    robot6axis_ctrled1/robot6axis/servo_2/servo_control/OperationMode AT 677 : INT := 0;
    robot6axis_ctrled1/robot6axis/servo_2/servo_control/StatusReady AT 253 : BOOL := true;
    robot6axis_ctrled1/robot6axis/servo_2/servo_control/StatusMove AT 254 : BOOL := false;
    robot6axis_ctrled1/robot6axis/servo_2/servo_control/StatusStand AT 255 : BOOL := false;
    robot6axis_ctrled1/robot6axis/servo_2/servo_control/ActualPositionMa AT 6703 : REAL := 0.0;
    robot6axis_ctrled1/robot6axis/servo_2/servo_control/ActualVelocity AT 6704 : REAL := 0.0;
    robot6axis_ctrled1/robot6axis/servo_2/servo_control/MaximumVelocity AT 6705 : REAL := 0.0;
    robot6axis_ctrled1/robot6axis/servo_2/servo_control/VelEnabled AT 256 : BOOL := false;
    robot6axis_ctrled1/robot6axis/servo_2/servo_control/VelCmd AT 257 : BOOL := false;
    robot6axis_ctrled1/robot6axis/servo_2/servo_control/PosEnabled AT 258 : BOOL := false;
    robot6axis_ctrled1/robot6axis/servo_2/servo_control/PosCmd AT 259 : BOOL := false;
    robot6axis_ctrled1/robot6axis/servo_2/servo_control/Position AT 6707 : REAL := 0.0;
    robot6axis_ctrled1/robot6axis/servo_2/servo_control/Speed AT 6706 : REAL := 0.0;
    robot6axis_ctrled1/robot6axis/servo_2/servo_control/ManualMode AT 678 : INT := 0;
    robot6axis_ctrled1/robot6axis/servo_2/servo_control/initDone AT 263 : BOOL := false;
    robot6axis_ctrled1/robot6axis/servo_2/servo_control/ActualPositionMa1 AT 6717 : REAL := 0.0;
    robot6axis_ctrled1/robot6axis/servo_2/servo_control/offsetAxToMa1 AT 6718 : REAL := 0.0;
    robot6axis_ctrled1/robot6axis/servo_2/servo_control/HOME_POSITION AT 6719 : REAL := 100.0;
    robot6axis_ctrled1/robot6axis/servo_2/servo_control/MANUAL_POSITION1 AT 6720 : REAL := 0.0;
    robot6axis_ctrled1/robot6axis/servo_2/servo_control/MANUAL_POSITION2 AT 6721 : REAL := 150.0;
    robot6axis_ctrled1/robot6axis/servo_2/servo_control/MANUAL_SPEED1 AT 6722 : REAL := -100.0;
    robot6axis_ctrled1/robot6axis/servo_2/servo_control/MANUAL_SPEED2 AT 6723 : REAL := 100.0;
    robot6axis_ctrled1/robot6axis/servo_2/servo_control/MANUAL_SPEED AT 6724 : REAL := 100.0;
    robot6axis_ctrled1/robot6axis/servo_2/servo_velocity/MoveVelEnable AT 256 : BOOL := false;
    robot6axis_ctrled1/robot6axis/servo_2/servo_velocity/MoveVelStart AT 257 : BOOL := false;
    robot6axis_ctrled1/robot6axis/servo_2/servo_velocity/MoveSpeed AT 6706 : REAL := 0.0;
    robot6axis_ctrled1/robot6axis/servo_2/servo_velocity/MoveAcceleration AT 86 : REAL := 100.0;
    robot6axis_ctrled1/robot6axis/servo_2/servo_velocity/MoveDeceleration AT 85 : REAL := 100.0;
    robot6axis_ctrled1/robot6axis/servo_2/servo_velocity/MAX_SPEED AT 6499 : REAL(0.0..3.4e+038) := 30.0;
    robot6axis_ctrled1/robot6axis/servo_2/servo_velocity/MAX_ACCEL AT 6498 : REAL(0.0..3.4e+038) := 1500.0;
    robot6axis_ctrled1/robot6axis/servo_2/servo_velocity/MAX_DECEL AT 6497 : REAL(0.0..3.4e+038) := 1500.0;
    robot6axis_ctrled1/robot6axis/servo_2/servo_velocity/MODULO_LENGTH AT 6496 : REAL := 0.0;
    robot6axis_ctrled1/robot6axis/servo_2/servo_velocity/status AT 661 : INT := 0;
    robot6axis_ctrled1/robot6axis/servo_2/servo_velocity/errorFlag AT 660 : INT := 0;
    robot6axis_ctrled1/robot6axis/servo_2/servo_velocity/MoveVelDone AT 225 : BOOL := false;
    robot6axis_ctrled1/robot6axis/servo_2/servo_velocity/ActualPositionAx AT 6502 : REAL := 0.0;
    robot6axis_ctrled1/robot6axis/servo_2/servo_velocity/ActualVelocity AT 6501 : REAL := 0.0;
    robot6axis_ctrled1/robot6axis/servo_2/servo_velocity/firstStep AT 264 : BOOL := true;
    robot6axis_ctrled1/robot6axis/servo_2/servo_velocity/stepDone AT 265 : BOOL := false;
    robot6axis_ctrled1/robot6axis/servo_2/servo_velocity/currentTime AT 6725 : REAL := 0.0;
    robot6axis_ctrled1/robot6axis/servo_2/servo_velocity/MoveSpeed1 AT 6726 : REAL := 0.0;
    robot6axis_ctrled1/robot6axis/servo_2/servo_velocity/acceleration AT 6727 : REAL := 0.0;
    robot6axis_ctrled1/robot6axis/servo_2/servo_velocity/deceleration AT 6728 : REAL := 0.0;
    robot6axis_ctrled1/robot6axis/servo_2/servo_velocity/orderSpeed AT 6729 : REAL := 0.0;
    robot6axis_ctrled1/robot6axis/servo_2/servo_velocity/endChangeSpeed AT 6730 : REAL := 0.0;
    robot6axis_ctrled1/robot6axis/servo_2/servo_velocity/accelDecelChangeSpeed AT 6731 : REAL := 0.0;
    robot6axis_ctrled1/robot6axis/servo_2/servo_velocity/ActualVelocity1 AT 6732 : REAL := 0.0;
    robot6axis_ctrled1/robot6axis/servo_2/servo_velocity/speedChanged AT 266 : BOOL := false;
    robot6axis_ctrled1/robot6axis/servo_2/servo_position/MoveAbsEnable AT 258 : BOOL := false;
    robot6axis_ctrled1/robot6axis/servo_2/servo_position/MoveAbsStart AT 259 : BOOL := false;
    robot6axis_ctrled1/robot6axis/servo_2/servo_position/MovePosition AT 6707 : REAL := 0.0;
    robot6axis_ctrled1/robot6axis/servo_2/servo_position/MoveSpeed AT 6706 : REAL := 0.0;
    robot6axis_ctrled1/robot6axis/servo_2/servo_position/MoveAcceleration AT 86 : REAL := 100.0;
    robot6axis_ctrled1/robot6axis/servo_2/servo_position/MoveDeceleration AT 85 : REAL := 100.0;
    robot6axis_ctrled1/robot6axis/servo_2/servo_position/MAX_SPEED AT 6499 : REAL(0.0..3.4e+038) := 30.0;
    robot6axis_ctrled1/robot6axis/servo_2/servo_position/MAX_ACCEL AT 6498 : REAL(0.0..3.4e+038) := 1500.0;
    robot6axis_ctrled1/robot6axis/servo_2/servo_position/MAX_DECEL AT 6497 : REAL(0.0..3.4e+038) := 1500.0;
    robot6axis_ctrled1/robot6axis/servo_2/servo_position/MODULO_LENGTH AT 6496 : REAL := 0.0;
    robot6axis_ctrled1/robot6axis/servo_2/servo_position/status AT 661 : INT := 0;
    robot6axis_ctrled1/robot6axis/servo_2/servo_position/errorFlag AT 660 : INT := 0;
    robot6axis_ctrled1/robot6axis/servo_2/servo_position/MoveAbsDone AT 224 : BOOL := false;
    robot6axis_ctrled1/robot6axis/servo_2/servo_position/ActualPositionAx AT 6502 : REAL := 0.0;
    robot6axis_ctrled1/robot6axis/servo_2/servo_position/ActualVelocity AT 6501 : REAL := 0.0;
    robot6axis_ctrled1/robot6axis/servo_2/servo_position/firstStep AT 267 : BOOL := true;
    robot6axis_ctrled1/robot6axis/servo_2/servo_position/stepDone AT 268 : BOOL := false;
    robot6axis_ctrled1/robot6axis/servo_2/servo_position/timeToStop AT 6733 : REAL := 0.0;
    robot6axis_ctrled1/robot6axis/servo_2/servo_position/distanceToStop AT 6734 : REAL := 0.0;
    robot6axis_ctrled1/robot6axis/servo_2/servo_position/distance AT 6735 : REAL := 0.0;
    robot6axis_ctrled1/robot6axis/servo_2/servo_position/currentTime AT 6736 : REAL := 0.0;
    robot6axis_ctrled1/robot6axis/servo_2/servo_position/currentSpeed1 AT 6737 : REAL := 0.0;
    robot6axis_ctrled1/robot6axis/servo_2/servo_position/targetPosition AT 6738 : REAL := 0.0;
    robot6axis_ctrled1/robot6axis/servo_2/servo_position/ActualPositionAx1 AT 6739 : REAL := 0.0;
    robot6axis_ctrled1/robot6axis/servo_2/servo_position/acceleration AT 6740 : REAL := 0.0;
    robot6axis_ctrled1/robot6axis/servo_2/servo_position/deceleration AT 6741 : REAL := 0.0;
    robot6axis_ctrled1/robot6axis/servo_2/servo_position/orderSpeed AT 6742 : REAL := 0.0;
    robot6axis_ctrled1/robot6axis/servo_2/servo_position/moveDirection AT 6743 : REAL := 0.0;
    robot6axis_ctrled1/robot6axis/servo_2/servo_position/moveDirection1 AT 6744 : REAL := 0.0;
    robot6axis_ctrled1/robot6axis/servo_2/servo_position/endChangeSpeed AT 6745 : REAL := 0.0;
    robot6axis_ctrled1/robot6axis/servo_2/servo_position/ActualVelocity1 AT 6746 : REAL := 0.0;
    robot6axis_ctrled1/robot6axis/arm2/armOrigin AT 6540 : ARRAY[1..3] OF REAL := [3(0.0)];
    robot6axis_ctrled1/robot6axis/arm2/overallArmQuatInput AT 6545 : ARRAY[1..4] OF REAL := [4(0.0)];
    robot6axis_ctrled1/robot6axis/arm2/structRotVector AT 149 : ARRAY[1..3] OF REAL := [2(0.0), 1.0];
    robot6axis_ctrled1/robot6axis/arm2/structRotDeg AT 148 : REAL := -90.0;
    robot6axis_ctrled1/robot6axis/arm2/driveRotVector AT 138 : ARRAY[1..3] OF REAL := [0.0, 1.0, 0.0];
    robot6axis_ctrled1/robot6axis/arm2/driveRotDeg AT 6551 : REAL := 0.0;
    robot6axis_ctrled1/robot6axis/arm2/ownRotDeg AT 6492 : REAL := 0.0;
    robot6axis_ctrled1/robot6axis/arm2/driveResizeLength AT 6491 : REAL := 0.0;
    robot6axis_ctrled1/robot6axis/arm2/functionActive AT 218 : BOOL := false;
    robot6axis_ctrled1/robot6axis/arm2/armExtrem AT 6552 : ARRAY[1..3] OF REAL := [3(0.0)];
    robot6axis_ctrled1/robot6axis/arm2/overallArmRotOutput AT 6557 : ARRAY[1..4] OF REAL := [4(0.0)];
    robot6axis_ctrled1/robot6axis/arm2/productId AT 659 : DINT := -1;
    robot6axis_ctrled1/robot6axis/arm2/status_act_prod AT 679 : DINT := 0;
    robot6axis_ctrled1/robot6axis/arm2/m11 AT 6747 : REAL := 127.321;
    robot6axis_ctrled1/robot6axis/arm2/m12 AT 6748 : REAL := 0.0;
    robot6axis_ctrled1/robot6axis/arm2/m13 AT 6749 : REAL := 0.0;
    robot6axis_ctrled1/robot6axis/arm2/m14 AT 6750 : REAL := 453.404;
    robot6axis_ctrled1/robot6axis/arm2/m21 AT 6751 : REAL := 0.0;
    robot6axis_ctrled1/robot6axis/arm2/m22 AT 6752 : REAL := 1.0;
    robot6axis_ctrled1/robot6axis/arm2/m23 AT 6753 : REAL := 0.0;
    robot6axis_ctrled1/robot6axis/arm2/m24 AT 6754 : REAL := 1.0;
    robot6axis_ctrled1/robot6axis/arm2/m31 AT 6755 : REAL := 0.0;
    robot6axis_ctrled1/robot6axis/arm2/m32 AT 6756 : REAL := 0.0;
    robot6axis_ctrled1/robot6axis/arm2/m33 AT 6757 : REAL := 35.3669;
    robot6axis_ctrled1/robot6axis/arm2/m34 AT 6758 : REAL := 213.705;
    robot6axis_ctrled1/robot6axis/arm2/m41 AT 6759 : REAL := 0.0;
    robot6axis_ctrled1/robot6axis/arm2/m42 AT 6760 : REAL := 0.0;
    robot6axis_ctrled1/robot6axis/arm2/m43 AT 6761 : REAL := 0.0;
    robot6axis_ctrled1/robot6axis/arm2/m44 AT 6762 : REAL := 1.0;
    robot6axis_ctrled1/robot6axis/arm2/armLengthCalc AT 6763 : REAL := 0.0;
    robot6axis_ctrled1/robot6axis/arm2/functionActiveLocale AT 269 : BOOL := false;
    robot6axis_ctrled1/robot6axis/arm2/product_id AT 680 : DINT := -1;
    robot6axis_ctrled1/robot6axis/arm2/arm_id AT 681 : DINT := -1;
    robot6axis_ctrled1/robot6axis/arm2/timeToGripParam AT 6764 : REAL := 0.15;
    robot6axis_ctrled1/robot6axis/arm2/armLength AT 6765 : REAL := 290.0;
    robot6axis_ctrled1/robot6axis/arm2/armWidth AT 6766 : REAL := 60.0;
    robot6axis_ctrled1/robot6axis/arm2/armHeight AT 6767 : REAL := 60.0;
    robot6axis_ctrled1/robot6axis/arm2/armType AT 682 : INT := 0;
    robot6axis_ctrled1/robot6axis/servo_3/status AT 658 : INT := 0;
    robot6axis_ctrled1/robot6axis/servo_3/errorFlag AT 657 : INT := 0;
    robot6axis_ctrled1/robot6axis/servo_3/ActualPositionAx1 AT 6490 : REAL := 0.0;
    robot6axis_ctrled1/robot6axis/servo_3/MoveVelDone1 AT 217 : BOOL := false;
    robot6axis_ctrled1/robot6axis/servo_3/ActualVelocity1 AT 6489 : REAL := 0.0;
    robot6axis_ctrled1/robot6axis/servo_3/MoveAbsDone1 AT 216 : BOOL := false;
    robot6axis_ctrled1/robot6axis/servo_3/HomeCmd AT 84 : BOOL := false;
    robot6axis_ctrled1/robot6axis/servo_3/MoveVelCmd AT 83 : BOOL := false;
    robot6axis_ctrled1/robot6axis/servo_3/MoveAbsCmd AT 82 : BOOL := false;
    robot6axis_ctrled1/robot6axis/servo_3/MoveVel1ManualCmd AT 81 : BOOL := false;
    robot6axis_ctrled1/robot6axis/servo_3/MoveVel2ManualCmd AT 80 : BOOL := false;
    robot6axis_ctrled1/robot6axis/servo_3/MoveAbs1ManualCmd AT 79 : BOOL := false;
    robot6axis_ctrled1/robot6axis/servo_3/MoveAbs2ManualCmd AT 78 : BOOL := false;
    robot6axis_ctrled1/robot6axis/servo_3/StopCmd AT 22 : BOOL := false;
    robot6axis_ctrled1/robot6axis/servo_3/MovePosition AT 83 : REAL := 0.0;
    robot6axis_ctrled1/robot6axis/servo_3/MoveSpeed AT 82 : REAL := 100.0;
    robot6axis_ctrled1/robot6axis/servo_3/MoveAcceleration AT 81 : REAL := 100.0;
    robot6axis_ctrled1/robot6axis/servo_3/MoveDeceleration AT 80 : REAL := 100.0;
    robot6axis_ctrled1/robot6axis/servo_3/offsetAxToMa AT 79 : REAL := 0.0;
    robot6axis_ctrled1/robot6axis/servo_3/PLC_StatusReady AT 50 : BOOL := true;
    robot6axis_ctrled1/robot6axis/servo_3/PLC_StatusMoved AT 49 : BOOL := false;
    robot6axis_ctrled1/robot6axis/servo_3/PLC_StatusStand AT 48 : BOOL := false;
    robot6axis_ctrled1/robot6axis/servo_3/PLC_ActualPositionAx AT 169 : REAL := 0.0;
    robot6axis_ctrled1/robot6axis/servo_3/PLC_ActualPositionMa AT 59 : REAL := 0.0;
    robot6axis_ctrled1/robot6axis/servo_3/PLC_ActualVelocity AT 58 : REAL := 0.0;
    robot6axis_ctrled1/robot6axis/servo_3/physicalPosInit AT 6488 : REAL := 0.0;
    robot6axis_ctrled1/robot6axis/servo_3/MAX_SPEED AT 6487 : REAL(0.0..3.4e+038) := 30.0;
    robot6axis_ctrled1/robot6axis/servo_3/MAX_ACCEL AT 6486 : REAL(0.0..3.4e+038) := 1500.0;
    robot6axis_ctrled1/robot6axis/servo_3/MAX_DECEL AT 6485 : REAL(0.0..3.4e+038) := 1500.0;
    robot6axis_ctrled1/robot6axis/servo_3/MODULO_LENGTH AT 6484 : REAL := 0.0;
    robot6axis_ctrled1/robot6axis/servo_3/StatusReady AT 215 : BOOL := true;
    robot6axis_ctrled1/robot6axis/servo_3/StatusMoved AT 214 : BOOL := false;
    robot6axis_ctrled1/robot6axis/servo_3/StatusStand AT 213 : BOOL := false;
    robot6axis_ctrled1/robot6axis/servo_3/ActualPositionAx AT 6563 : REAL := 0.0;
    robot6axis_ctrled1/robot6axis/servo_3/ActualPositionMa AT 6483 : REAL := 0.0;
    robot6axis_ctrled1/robot6axis/servo_3/ActualVelocity AT 49 : REAL := 0.0;
    robot6axis_ctrled1/robot6axis/servo_3/MaximumVelocity AT 6482 : REAL := 0.0;
    robot6axis_ctrled1/robot6axis/servo_3/StatusPosIncrease AT 212 : BOOL := false;
    robot6axis_ctrled1/robot6axis/servo_3/StatusPosDecrease AT 211 : BOOL := false;
    robot6axis_ctrled1/robot6axis/servo_3/displayJauge AT 6481 : REAL := 0.0;
    robot6axis_ctrled1/robot6axis/servo_3/servo_mode/PLC_StatusReady AT 50 : BOOL := true;
    robot6axis_ctrled1/robot6axis/servo_3/servo_mode/PLC_StatusMoved AT 49 : BOOL := false;
    robot6axis_ctrled1/robot6axis/servo_3/servo_mode/PLC_StatusStand AT 48 : BOOL := false;
    robot6axis_ctrled1/robot6axis/servo_3/servo_mode/PLC_ActualPositionAx AT 169 : REAL := 0.0;
    robot6axis_ctrled1/robot6axis/servo_3/servo_mode/PLC_ActualPositionMa AT 59 : REAL := 0.0;
    robot6axis_ctrled1/robot6axis/servo_3/servo_mode/PLC_ActualVelocity AT 58 : REAL := 0.0;
    robot6axis_ctrled1/robot6axis/servo_3/servo_mode/StatusReady AT 270 : BOOL := true;
    robot6axis_ctrled1/robot6axis/servo_3/servo_mode/StatusMoved AT 271 : BOOL := false;
    robot6axis_ctrled1/robot6axis/servo_3/servo_mode/StatusStand AT 272 : BOOL := false;
    robot6axis_ctrled1/robot6axis/servo_3/servo_mode/ActualPositionMa AT 6768 : REAL := 0.0;
    robot6axis_ctrled1/robot6axis/servo_3/servo_mode/ActualVelocity AT 6769 : REAL := 0.0;
    robot6axis_ctrled1/robot6axis/servo_3/servo_mode/MaximumVelocity AT 6770 : REAL := 0.0;
    robot6axis_ctrled1/robot6axis/servo_3/servo_mode/physicalPosInit AT 6488 : REAL := 0.0;
    robot6axis_ctrled1/robot6axis/servo_3/servo_mode/ActualPositionAx AT 6490 : REAL := 0.0;
    robot6axis_ctrled1/robot6axis/servo_3/servo_mode/StatusReady_o AT 215 : BOOL := true;
    robot6axis_ctrled1/robot6axis/servo_3/servo_mode/StatusMoved_o AT 214 : BOOL := false;
    robot6axis_ctrled1/robot6axis/servo_3/servo_mode/StatusStand_o AT 213 : BOOL := false;
    robot6axis_ctrled1/robot6axis/servo_3/servo_mode/ActualPositionAx_o AT 6563 : REAL := 0.0;
    robot6axis_ctrled1/robot6axis/servo_3/servo_mode/ActualPositionMa_o AT 6483 : REAL := 0.0;
    robot6axis_ctrled1/robot6axis/servo_3/servo_mode/ActualVelocity_o AT 49 : REAL := 0.0;
    robot6axis_ctrled1/robot6axis/servo_3/servo_mode/MaximumVelocity_o AT 6482 : REAL := 0.0;
    robot6axis_ctrled1/robot6axis/servo_3/servo_mode/StatusPosIncrease_o AT 212 : BOOL := false;
    robot6axis_ctrled1/robot6axis/servo_3/servo_mode/StatusPosDecrease_o AT 211 : BOOL := false;
    robot6axis_ctrled1/robot6axis/servo_3/servo_mode/displayJauge_o AT 6481 : REAL := 0.0;
    robot6axis_ctrled1/robot6axis/servo_3/servo_mode/PLCMode AT 277 : BOOL := false;
    robot6axis_ctrled1/robot6axis/servo_3/servo_mode/PLCMode1 AT 278 : BOOL := false;
    robot6axis_ctrled1/robot6axis/servo_3/servo_mode/initDone AT 279 : BOOL := false;
    robot6axis_ctrled1/robot6axis/servo_3/servo_mode/displayPosMin AT 6773 : REAL := 0.0;
    robot6axis_ctrled1/robot6axis/servo_3/servo_mode/displayPosMax AT 6774 : REAL := 0.0;
    robot6axis_ctrled1/robot6axis/servo_3/servo_mode/PLC_ActualPositionAx1 AT 6775 : REAL := 0.0;
    robot6axis_ctrled1/robot6axis/servo_3/servo_mode/PLC_ActualVelocity1 AT 6776 : REAL := 0.0;
    robot6axis_ctrled1/robot6axis/servo_3/servo_mode/ActualPositionAx1 AT 6777 : REAL := 0.0;
    robot6axis_ctrled1/robot6axis/servo_3/servo_mode/ActualVelocity1 AT 6778 : REAL := 0.0;
    robot6axis_ctrled1/robot6axis/servo_3/servo_mode/offsetAxToMa AT 6779 : REAL := 0.0;
    robot6axis_ctrled1/robot6axis/servo_3/servo_mode/offsetAxToMa1 AT 6780 : REAL := 0.0;
    robot6axis_ctrled1/robot6axis/servo_3/servo_mode/ActualPositionMa_o1 AT 6781 : REAL := 0.0;
    robot6axis_ctrled1/robot6axis/servo_3/servo_control/HomeCmd AT 84 : BOOL := false;
    robot6axis_ctrled1/robot6axis/servo_3/servo_control/MoveVelCmd AT 83 : BOOL := false;
    robot6axis_ctrled1/robot6axis/servo_3/servo_control/MoveAbsCmd AT 82 : BOOL := false;
    robot6axis_ctrled1/robot6axis/servo_3/servo_control/MoveVel1ManualCmd AT 81 : BOOL := false;
    robot6axis_ctrled1/robot6axis/servo_3/servo_control/MoveVel2ManualCmd AT 80 : BOOL := false;
    robot6axis_ctrled1/robot6axis/servo_3/servo_control/MoveAbs1ManualCmd AT 79 : BOOL := false;
    robot6axis_ctrled1/robot6axis/servo_3/servo_control/MoveAbs2ManualCmd AT 78 : BOOL := false;
    robot6axis_ctrled1/robot6axis/servo_3/servo_control/StopCmd AT 22 : BOOL := false;
    robot6axis_ctrled1/robot6axis/servo_3/servo_control/MovePosition AT 83 : REAL := 0.0;
    robot6axis_ctrled1/robot6axis/servo_3/servo_control/MoveSpeed AT 82 : REAL := 100.0;
    robot6axis_ctrled1/robot6axis/servo_3/servo_control/MoveAcceleration AT 81 : REAL := 100.0;
    robot6axis_ctrled1/robot6axis/servo_3/servo_control/MoveDeceleration AT 80 : REAL := 100.0;
    robot6axis_ctrled1/robot6axis/servo_3/servo_control/offsetAxToMa AT 79 : REAL := 0.0;
    robot6axis_ctrled1/robot6axis/servo_3/servo_control/physicalPosInit AT 6488 : REAL := 0.0;
    robot6axis_ctrled1/robot6axis/servo_3/servo_control/MAX_SPEED AT 6487 : REAL(0.0..3.4e+038) := 30.0;
    robot6axis_ctrled1/robot6axis/servo_3/servo_control/status AT 658 : INT := 0;
    robot6axis_ctrled1/robot6axis/servo_3/servo_control/errorFlag AT 657 : INT := 0;
    robot6axis_ctrled1/robot6axis/servo_3/servo_control/IOActualPositionAx AT 6490 : REAL := 0.0;
    robot6axis_ctrled1/robot6axis/servo_3/servo_control/IOVelDone AT 217 : BOOL := false;
    robot6axis_ctrled1/robot6axis/servo_3/servo_control/IOAbsDone AT 216 : BOOL := false;
    robot6axis_ctrled1/robot6axis/servo_3/servo_control/IOActualVelocity AT 6489 : REAL := 0.0;
    robot6axis_ctrled1/robot6axis/servo_3/servo_control/OperationMode AT 683 : INT := 0;
    robot6axis_ctrled1/robot6axis/servo_3/servo_control/StatusReady AT 270 : BOOL := true;
    robot6axis_ctrled1/robot6axis/servo_3/servo_control/StatusMove AT 271 : BOOL := false;
    robot6axis_ctrled1/robot6axis/servo_3/servo_control/StatusStand AT 272 : BOOL := false;
    robot6axis_ctrled1/robot6axis/servo_3/servo_control/ActualPositionMa AT 6768 : REAL := 0.0;
    robot6axis_ctrled1/robot6axis/servo_3/servo_control/ActualVelocity AT 6769 : REAL := 0.0;
    robot6axis_ctrled1/robot6axis/servo_3/servo_control/MaximumVelocity AT 6770 : REAL := 0.0;
    robot6axis_ctrled1/robot6axis/servo_3/servo_control/VelEnabled AT 273 : BOOL := false;
    robot6axis_ctrled1/robot6axis/servo_3/servo_control/VelCmd AT 274 : BOOL := false;
    robot6axis_ctrled1/robot6axis/servo_3/servo_control/PosEnabled AT 275 : BOOL := false;
    robot6axis_ctrled1/robot6axis/servo_3/servo_control/PosCmd AT 276 : BOOL := false;
    robot6axis_ctrled1/robot6axis/servo_3/servo_control/Position AT 6772 : REAL := 0.0;
    robot6axis_ctrled1/robot6axis/servo_3/servo_control/Speed AT 6771 : REAL := 0.0;
    robot6axis_ctrled1/robot6axis/servo_3/servo_control/ManualMode AT 684 : INT := 0;
    robot6axis_ctrled1/robot6axis/servo_3/servo_control/initDone AT 280 : BOOL := false;
    robot6axis_ctrled1/robot6axis/servo_3/servo_control/ActualPositionMa1 AT 6782 : REAL := 0.0;
    robot6axis_ctrled1/robot6axis/servo_3/servo_control/offsetAxToMa1 AT 6783 : REAL := 0.0;
    robot6axis_ctrled1/robot6axis/servo_3/servo_control/HOME_POSITION AT 6784 : REAL := 100.0;
    robot6axis_ctrled1/robot6axis/servo_3/servo_control/MANUAL_POSITION1 AT 6785 : REAL := 0.0;
    robot6axis_ctrled1/robot6axis/servo_3/servo_control/MANUAL_POSITION2 AT 6786 : REAL := 150.0;
    robot6axis_ctrled1/robot6axis/servo_3/servo_control/MANUAL_SPEED1 AT 6787 : REAL := -100.0;
    robot6axis_ctrled1/robot6axis/servo_3/servo_control/MANUAL_SPEED2 AT 6788 : REAL := 100.0;
    robot6axis_ctrled1/robot6axis/servo_3/servo_control/MANUAL_SPEED AT 6789 : REAL := 100.0;
    robot6axis_ctrled1/robot6axis/servo_3/servo_velocity/MoveVelEnable AT 273 : BOOL := false;
    robot6axis_ctrled1/robot6axis/servo_3/servo_velocity/MoveVelStart AT 274 : BOOL := false;
    robot6axis_ctrled1/robot6axis/servo_3/servo_velocity/MoveSpeed AT 6771 : REAL := 0.0;
    robot6axis_ctrled1/robot6axis/servo_3/servo_velocity/MoveAcceleration AT 81 : REAL := 100.0;
    robot6axis_ctrled1/robot6axis/servo_3/servo_velocity/MoveDeceleration AT 80 : REAL := 100.0;
    robot6axis_ctrled1/robot6axis/servo_3/servo_velocity/MAX_SPEED AT 6487 : REAL(0.0..3.4e+038) := 30.0;
    robot6axis_ctrled1/robot6axis/servo_3/servo_velocity/MAX_ACCEL AT 6486 : REAL(0.0..3.4e+038) := 1500.0;
    robot6axis_ctrled1/robot6axis/servo_3/servo_velocity/MAX_DECEL AT 6485 : REAL(0.0..3.4e+038) := 1500.0;
    robot6axis_ctrled1/robot6axis/servo_3/servo_velocity/MODULO_LENGTH AT 6484 : REAL := 0.0;
    robot6axis_ctrled1/robot6axis/servo_3/servo_velocity/status AT 658 : INT := 0;
    robot6axis_ctrled1/robot6axis/servo_3/servo_velocity/errorFlag AT 657 : INT := 0;
    robot6axis_ctrled1/robot6axis/servo_3/servo_velocity/MoveVelDone AT 217 : BOOL := false;
    robot6axis_ctrled1/robot6axis/servo_3/servo_velocity/ActualPositionAx AT 6490 : REAL := 0.0;
    robot6axis_ctrled1/robot6axis/servo_3/servo_velocity/ActualVelocity AT 6489 : REAL := 0.0;
    robot6axis_ctrled1/robot6axis/servo_3/servo_velocity/firstStep AT 281 : BOOL := true;
    robot6axis_ctrled1/robot6axis/servo_3/servo_velocity/stepDone AT 282 : BOOL := false;
    robot6axis_ctrled1/robot6axis/servo_3/servo_velocity/currentTime AT 6790 : REAL := 0.0;
    robot6axis_ctrled1/robot6axis/servo_3/servo_velocity/MoveSpeed1 AT 6791 : REAL := 0.0;
    robot6axis_ctrled1/robot6axis/servo_3/servo_velocity/acceleration AT 6792 : REAL := 0.0;
    robot6axis_ctrled1/robot6axis/servo_3/servo_velocity/deceleration AT 6793 : REAL := 0.0;
    robot6axis_ctrled1/robot6axis/servo_3/servo_velocity/orderSpeed AT 6794 : REAL := 0.0;
    robot6axis_ctrled1/robot6axis/servo_3/servo_velocity/endChangeSpeed AT 6795 : REAL := 0.0;
    robot6axis_ctrled1/robot6axis/servo_3/servo_velocity/accelDecelChangeSpeed AT 6796 : REAL := 0.0;
    robot6axis_ctrled1/robot6axis/servo_3/servo_velocity/ActualVelocity1 AT 6797 : REAL := 0.0;
    robot6axis_ctrled1/robot6axis/servo_3/servo_velocity/speedChanged AT 283 : BOOL := false;
    robot6axis_ctrled1/robot6axis/servo_3/servo_position/MoveAbsEnable AT 275 : BOOL := false;
    robot6axis_ctrled1/robot6axis/servo_3/servo_position/MoveAbsStart AT 276 : BOOL := false;
    robot6axis_ctrled1/robot6axis/servo_3/servo_position/MovePosition AT 6772 : REAL := 0.0;
    robot6axis_ctrled1/robot6axis/servo_3/servo_position/MoveSpeed AT 6771 : REAL := 0.0;
    robot6axis_ctrled1/robot6axis/servo_3/servo_position/MoveAcceleration AT 81 : REAL := 100.0;
    robot6axis_ctrled1/robot6axis/servo_3/servo_position/MoveDeceleration AT 80 : REAL := 100.0;
    robot6axis_ctrled1/robot6axis/servo_3/servo_position/MAX_SPEED AT 6487 : REAL(0.0..3.4e+038) := 30.0;
    robot6axis_ctrled1/robot6axis/servo_3/servo_position/MAX_ACCEL AT 6486 : REAL(0.0..3.4e+038) := 1500.0;
    robot6axis_ctrled1/robot6axis/servo_3/servo_position/MAX_DECEL AT 6485 : REAL(0.0..3.4e+038) := 1500.0;
    robot6axis_ctrled1/robot6axis/servo_3/servo_position/MODULO_LENGTH AT 6484 : REAL := 0.0;
    robot6axis_ctrled1/robot6axis/servo_3/servo_position/status AT 658 : INT := 0;
    robot6axis_ctrled1/robot6axis/servo_3/servo_position/errorFlag AT 657 : INT := 0;
    robot6axis_ctrled1/robot6axis/servo_3/servo_position/MoveAbsDone AT 216 : BOOL := false;
    robot6axis_ctrled1/robot6axis/servo_3/servo_position/ActualPositionAx AT 6490 : REAL := 0.0;
    robot6axis_ctrled1/robot6axis/servo_3/servo_position/ActualVelocity AT 6489 : REAL := 0.0;
    robot6axis_ctrled1/robot6axis/servo_3/servo_position/firstStep AT 284 : BOOL := true;
    robot6axis_ctrled1/robot6axis/servo_3/servo_position/stepDone AT 285 : BOOL := false;
    robot6axis_ctrled1/robot6axis/servo_3/servo_position/timeToStop AT 6798 : REAL := 0.0;
    robot6axis_ctrled1/robot6axis/servo_3/servo_position/distanceToStop AT 6799 : REAL := 0.0;
    robot6axis_ctrled1/robot6axis/servo_3/servo_position/distance AT 6800 : REAL := 0.0;
    robot6axis_ctrled1/robot6axis/servo_3/servo_position/currentTime AT 6801 : REAL := 0.0;
    robot6axis_ctrled1/robot6axis/servo_3/servo_position/currentSpeed1 AT 6802 : REAL := 0.0;
    robot6axis_ctrled1/robot6axis/servo_3/servo_position/targetPosition AT 6803 : REAL := 0.0;
    robot6axis_ctrled1/robot6axis/servo_3/servo_position/ActualPositionAx1 AT 6804 : REAL := 0.0;
    robot6axis_ctrled1/robot6axis/servo_3/servo_position/acceleration AT 6805 : REAL := 0.0;
    robot6axis_ctrled1/robot6axis/servo_3/servo_position/deceleration AT 6806 : REAL := 0.0;
    robot6axis_ctrled1/robot6axis/servo_3/servo_position/orderSpeed AT 6807 : REAL := 0.0;
    robot6axis_ctrled1/robot6axis/servo_3/servo_position/moveDirection AT 6808 : REAL := 0.0;
    robot6axis_ctrled1/robot6axis/servo_3/servo_position/moveDirection1 AT 6809 : REAL := 0.0;
    robot6axis_ctrled1/robot6axis/servo_3/servo_position/endChangeSpeed AT 6810 : REAL := 0.0;
    robot6axis_ctrled1/robot6axis/servo_3/servo_position/ActualVelocity1 AT 6811 : REAL := 0.0;
    robot6axis_ctrled1/robot6axis/arm3/armOrigin AT 6552 : ARRAY[1..3] OF REAL := [3(0.0)];
    robot6axis_ctrled1/robot6axis/arm3/overallArmQuatInput AT 6557 : ARRAY[1..4] OF REAL := [4(0.0)];
    robot6axis_ctrled1/robot6axis/arm3/structRotVector AT 6476 : ARRAY[1..3] OF REAL := [2(0.0), 1.0];
    robot6axis_ctrled1/robot6axis/arm3/structRotDeg AT 6475 : REAL := 0.0;
    robot6axis_ctrled1/robot6axis/arm3/driveRotVector AT 133 : ARRAY[1..3] OF REAL := [0.0, 1.0, 0.0];
    robot6axis_ctrled1/robot6axis/arm3/driveRotDeg AT 6563 : REAL := 0.0;
    robot6axis_ctrled1/robot6axis/arm3/ownRotDeg AT 6474 : REAL := 0.0;
    robot6axis_ctrled1/robot6axis/arm3/driveResizeLength AT 6473 : REAL := 0.0;
    robot6axis_ctrled1/robot6axis/arm3/functionActive AT 210 : BOOL := false;
    robot6axis_ctrled1/robot6axis/arm3/armExtrem AT 6564 : ARRAY[1..3] OF REAL := [3(0.0)];
    robot6axis_ctrled1/robot6axis/arm3/overallArmRotOutput AT 6569 : ARRAY[1..4] OF REAL := [4(0.0)];
    robot6axis_ctrled1/robot6axis/arm3/productId AT 656 : DINT := -1;
    robot6axis_ctrled1/robot6axis/arm3/status_act_prod AT 685 : DINT := 0;
    robot6axis_ctrled1/robot6axis/arm3/m11 AT 6812 : REAL := 127.321;
    robot6axis_ctrled1/robot6axis/arm3/m12 AT 6813 : REAL := 0.0;
    robot6axis_ctrled1/robot6axis/arm3/m13 AT 6814 : REAL := 0.0;
    robot6axis_ctrled1/robot6axis/arm3/m14 AT 6815 : REAL := 456.587;
    robot6axis_ctrled1/robot6axis/arm3/m21 AT 6816 : REAL := 0.0;
    robot6axis_ctrled1/robot6axis/arm3/m22 AT 6817 : REAL := 1.0;
    robot6axis_ctrled1/robot6axis/arm3/m23 AT 6818 : REAL := 0.0;
    robot6axis_ctrled1/robot6axis/arm3/m24 AT 6819 : REAL := 1.0;
    robot6axis_ctrled1/robot6axis/arm3/m31 AT 6820 : REAL := 0.0;
    robot6axis_ctrled1/robot6axis/arm3/m32 AT 6821 : REAL := 0.0;
    robot6axis_ctrled1/robot6axis/arm3/m33 AT 6822 : REAL := 35.3669;
    robot6axis_ctrled1/robot6axis/arm3/m34 AT 6823 : REAL := 159.24;
    robot6axis_ctrled1/robot6axis/arm3/m41 AT 6824 : REAL := 0.0;
    robot6axis_ctrled1/robot6axis/arm3/m42 AT 6825 : REAL := 0.0;
    robot6axis_ctrled1/robot6axis/arm3/m43 AT 6826 : REAL := 0.0;
    robot6axis_ctrled1/robot6axis/arm3/m44 AT 6827 : REAL := 1.0;
    robot6axis_ctrled1/robot6axis/arm3/armLengthCalc AT 6828 : REAL := 0.0;
    robot6axis_ctrled1/robot6axis/arm3/functionActiveLocale AT 286 : BOOL := false;
    robot6axis_ctrled1/robot6axis/arm3/product_id AT 686 : DINT := -1;
    robot6axis_ctrled1/robot6axis/arm3/arm_id AT 687 : DINT := -1;
    robot6axis_ctrled1/robot6axis/arm3/timeToGripParam AT 6829 : REAL := 0.15;
    robot6axis_ctrled1/robot6axis/arm3/armLength AT 6830 : REAL := 108.0;
    robot6axis_ctrled1/robot6axis/arm3/armWidth AT 6831 : REAL := 60.0;
    robot6axis_ctrled1/robot6axis/arm3/armHeight AT 6832 : REAL := 60.0;
    robot6axis_ctrled1/robot6axis/arm3/armType AT 688 : INT := 0;
    robot6axis_ctrled1/robot6axis/servo_4/status AT 655 : INT := 0;
    robot6axis_ctrled1/robot6axis/servo_4/errorFlag AT 654 : INT := 0;
    robot6axis_ctrled1/robot6axis/servo_4/ActualPositionAx1 AT 6472 : REAL := 0.0;
    robot6axis_ctrled1/robot6axis/servo_4/MoveVelDone1 AT 209 : BOOL := false;
    robot6axis_ctrled1/robot6axis/servo_4/ActualVelocity1 AT 6471 : REAL := 0.0;
    robot6axis_ctrled1/robot6axis/servo_4/MoveAbsDone1 AT 208 : BOOL := false;
    robot6axis_ctrled1/robot6axis/servo_4/HomeCmd AT 77 : BOOL := false;
    robot6axis_ctrled1/robot6axis/servo_4/MoveVelCmd AT 76 : BOOL := false;
    robot6axis_ctrled1/robot6axis/servo_4/MoveAbsCmd AT 75 : BOOL := false;
    robot6axis_ctrled1/robot6axis/servo_4/MoveVel1ManualCmd AT 74 : BOOL := false;
    robot6axis_ctrled1/robot6axis/servo_4/MoveVel2ManualCmd AT 73 : BOOL := false;
    robot6axis_ctrled1/robot6axis/servo_4/MoveAbs1ManualCmd AT 72 : BOOL := false;
    robot6axis_ctrled1/robot6axis/servo_4/MoveAbs2ManualCmd AT 71 : BOOL := false;
    robot6axis_ctrled1/robot6axis/servo_4/StopCmd AT 22 : BOOL := false;
    robot6axis_ctrled1/robot6axis/servo_4/MovePosition AT 78 : REAL := 0.0;
    robot6axis_ctrled1/robot6axis/servo_4/MoveSpeed AT 77 : REAL := 100.0;
    robot6axis_ctrled1/robot6axis/servo_4/MoveAcceleration AT 76 : REAL := 100.0;
    robot6axis_ctrled1/robot6axis/servo_4/MoveDeceleration AT 75 : REAL := 100.0;
    robot6axis_ctrled1/robot6axis/servo_4/offsetAxToMa AT 74 : REAL := 0.0;
    robot6axis_ctrled1/robot6axis/servo_4/PLC_StatusReady AT 47 : BOOL := true;
    robot6axis_ctrled1/robot6axis/servo_4/PLC_StatusMoved AT 46 : BOOL := false;
    robot6axis_ctrled1/robot6axis/servo_4/PLC_StatusStand AT 45 : BOOL := false;
    robot6axis_ctrled1/robot6axis/servo_4/PLC_ActualPositionAx AT 170 : REAL := 0.0;
    robot6axis_ctrled1/robot6axis/servo_4/PLC_ActualPositionMa AT 57 : REAL := 0.0;
    robot6axis_ctrled1/robot6axis/servo_4/PLC_ActualVelocity AT 56 : REAL := 0.0;
    robot6axis_ctrled1/robot6axis/servo_4/physicalPosInit AT 6470 : REAL := 0.0;
    robot6axis_ctrled1/robot6axis/servo_4/MAX_SPEED AT 6469 : REAL(0.0..3.4e+038) := 30.0;
    robot6axis_ctrled1/robot6axis/servo_4/MAX_ACCEL AT 6468 : REAL(0.0..3.4e+038) := 1500.0;
    robot6axis_ctrled1/robot6axis/servo_4/MAX_DECEL AT 6467 : REAL(0.0..3.4e+038) := 1500.0;
    robot6axis_ctrled1/robot6axis/servo_4/MODULO_LENGTH AT 6466 : REAL := 0.0;
    robot6axis_ctrled1/robot6axis/servo_4/StatusReady AT 207 : BOOL := true;
    robot6axis_ctrled1/robot6axis/servo_4/StatusMoved AT 206 : BOOL := false;
    robot6axis_ctrled1/robot6axis/servo_4/StatusStand AT 205 : BOOL := false;
    robot6axis_ctrled1/robot6axis/servo_4/ActualPositionAx AT 6575 : REAL := 0.0;
    robot6axis_ctrled1/robot6axis/servo_4/ActualPositionMa AT 6465 : REAL := 0.0;
    robot6axis_ctrled1/robot6axis/servo_4/ActualVelocity AT 48 : REAL := 0.0;
    robot6axis_ctrled1/robot6axis/servo_4/MaximumVelocity AT 6464 : REAL := 0.0;
    robot6axis_ctrled1/robot6axis/servo_4/StatusPosIncrease AT 204 : BOOL := false;
    robot6axis_ctrled1/robot6axis/servo_4/StatusPosDecrease AT 203 : BOOL := false;
    robot6axis_ctrled1/robot6axis/servo_4/displayJauge AT 6463 : REAL := 0.0;
    robot6axis_ctrled1/robot6axis/servo_4/servo_mode/PLC_StatusReady AT 47 : BOOL := true;
    robot6axis_ctrled1/robot6axis/servo_4/servo_mode/PLC_StatusMoved AT 46 : BOOL := false;
    robot6axis_ctrled1/robot6axis/servo_4/servo_mode/PLC_StatusStand AT 45 : BOOL := false;
    robot6axis_ctrled1/robot6axis/servo_4/servo_mode/PLC_ActualPositionAx AT 170 : REAL := 0.0;
    robot6axis_ctrled1/robot6axis/servo_4/servo_mode/PLC_ActualPositionMa AT 57 : REAL := 0.0;
    robot6axis_ctrled1/robot6axis/servo_4/servo_mode/PLC_ActualVelocity AT 56 : REAL := 0.0;
    robot6axis_ctrled1/robot6axis/servo_4/servo_mode/StatusReady AT 287 : BOOL := true;
    robot6axis_ctrled1/robot6axis/servo_4/servo_mode/StatusMoved AT 288 : BOOL := false;
    robot6axis_ctrled1/robot6axis/servo_4/servo_mode/StatusStand AT 289 : BOOL := false;
    robot6axis_ctrled1/robot6axis/servo_4/servo_mode/ActualPositionMa AT 6833 : REAL := 0.0;
    robot6axis_ctrled1/robot6axis/servo_4/servo_mode/ActualVelocity AT 6834 : REAL := 0.0;
    robot6axis_ctrled1/robot6axis/servo_4/servo_mode/MaximumVelocity AT 6835 : REAL := 0.0;
    robot6axis_ctrled1/robot6axis/servo_4/servo_mode/physicalPosInit AT 6470 : REAL := 0.0;
    robot6axis_ctrled1/robot6axis/servo_4/servo_mode/ActualPositionAx AT 6472 : REAL := 0.0;
    robot6axis_ctrled1/robot6axis/servo_4/servo_mode/StatusReady_o AT 207 : BOOL := true;
    robot6axis_ctrled1/robot6axis/servo_4/servo_mode/StatusMoved_o AT 206 : BOOL := false;
    robot6axis_ctrled1/robot6axis/servo_4/servo_mode/StatusStand_o AT 205 : BOOL := false;
    robot6axis_ctrled1/robot6axis/servo_4/servo_mode/ActualPositionAx_o AT 6575 : REAL := 0.0;
    robot6axis_ctrled1/robot6axis/servo_4/servo_mode/ActualPositionMa_o AT 6465 : REAL := 0.0;
    robot6axis_ctrled1/robot6axis/servo_4/servo_mode/ActualVelocity_o AT 48 : REAL := 0.0;
    robot6axis_ctrled1/robot6axis/servo_4/servo_mode/MaximumVelocity_o AT 6464 : REAL := 0.0;
    robot6axis_ctrled1/robot6axis/servo_4/servo_mode/StatusPosIncrease_o AT 204 : BOOL := false;
    robot6axis_ctrled1/robot6axis/servo_4/servo_mode/StatusPosDecrease_o AT 203 : BOOL := false;
    robot6axis_ctrled1/robot6axis/servo_4/servo_mode/displayJauge_o AT 6463 : REAL := 0.0;
    robot6axis_ctrled1/robot6axis/servo_4/servo_mode/PLCMode AT 294 : BOOL := false;
    robot6axis_ctrled1/robot6axis/servo_4/servo_mode/PLCMode1 AT 295 : BOOL := false;
    robot6axis_ctrled1/robot6axis/servo_4/servo_mode/initDone AT 296 : BOOL := false;
    robot6axis_ctrled1/robot6axis/servo_4/servo_mode/displayPosMin AT 6838 : REAL := 0.0;
    robot6axis_ctrled1/robot6axis/servo_4/servo_mode/displayPosMax AT 6839 : REAL := 0.0;
    robot6axis_ctrled1/robot6axis/servo_4/servo_mode/PLC_ActualPositionAx1 AT 6840 : REAL := 0.0;
    robot6axis_ctrled1/robot6axis/servo_4/servo_mode/PLC_ActualVelocity1 AT 6841 : REAL := 0.0;
    robot6axis_ctrled1/robot6axis/servo_4/servo_mode/ActualPositionAx1 AT 6842 : REAL := 0.0;
    robot6axis_ctrled1/robot6axis/servo_4/servo_mode/ActualVelocity1 AT 6843 : REAL := 0.0;
    robot6axis_ctrled1/robot6axis/servo_4/servo_mode/offsetAxToMa AT 6844 : REAL := 0.0;
    robot6axis_ctrled1/robot6axis/servo_4/servo_mode/offsetAxToMa1 AT 6845 : REAL := 0.0;
    robot6axis_ctrled1/robot6axis/servo_4/servo_mode/ActualPositionMa_o1 AT 6846 : REAL := 0.0;
    robot6axis_ctrled1/robot6axis/servo_4/servo_control/HomeCmd AT 77 : BOOL := false;
    robot6axis_ctrled1/robot6axis/servo_4/servo_control/MoveVelCmd AT 76 : BOOL := false;
    robot6axis_ctrled1/robot6axis/servo_4/servo_control/MoveAbsCmd AT 75 : BOOL := false;
    robot6axis_ctrled1/robot6axis/servo_4/servo_control/MoveVel1ManualCmd AT 74 : BOOL := false;
    robot6axis_ctrled1/robot6axis/servo_4/servo_control/MoveVel2ManualCmd AT 73 : BOOL := false;
    robot6axis_ctrled1/robot6axis/servo_4/servo_control/MoveAbs1ManualCmd AT 72 : BOOL := false;
    robot6axis_ctrled1/robot6axis/servo_4/servo_control/MoveAbs2ManualCmd AT 71 : BOOL := false;
    robot6axis_ctrled1/robot6axis/servo_4/servo_control/StopCmd AT 22 : BOOL := false;
    robot6axis_ctrled1/robot6axis/servo_4/servo_control/MovePosition AT 78 : REAL := 0.0;
    robot6axis_ctrled1/robot6axis/servo_4/servo_control/MoveSpeed AT 77 : REAL := 100.0;
    robot6axis_ctrled1/robot6axis/servo_4/servo_control/MoveAcceleration AT 76 : REAL := 100.0;
    robot6axis_ctrled1/robot6axis/servo_4/servo_control/MoveDeceleration AT 75 : REAL := 100.0;
    robot6axis_ctrled1/robot6axis/servo_4/servo_control/offsetAxToMa AT 74 : REAL := 0.0;
    robot6axis_ctrled1/robot6axis/servo_4/servo_control/physicalPosInit AT 6470 : REAL := 0.0;
    robot6axis_ctrled1/robot6axis/servo_4/servo_control/MAX_SPEED AT 6469 : REAL(0.0..3.4e+038) := 30.0;
    robot6axis_ctrled1/robot6axis/servo_4/servo_control/status AT 655 : INT := 0;
    robot6axis_ctrled1/robot6axis/servo_4/servo_control/errorFlag AT 654 : INT := 0;
    robot6axis_ctrled1/robot6axis/servo_4/servo_control/IOActualPositionAx AT 6472 : REAL := 0.0;
    robot6axis_ctrled1/robot6axis/servo_4/servo_control/IOVelDone AT 209 : BOOL := false;
    robot6axis_ctrled1/robot6axis/servo_4/servo_control/IOAbsDone AT 208 : BOOL := false;
    robot6axis_ctrled1/robot6axis/servo_4/servo_control/IOActualVelocity AT 6471 : REAL := 0.0;
    robot6axis_ctrled1/robot6axis/servo_4/servo_control/OperationMode AT 689 : INT := 0;
    robot6axis_ctrled1/robot6axis/servo_4/servo_control/StatusReady AT 287 : BOOL := true;
    robot6axis_ctrled1/robot6axis/servo_4/servo_control/StatusMove AT 288 : BOOL := false;
    robot6axis_ctrled1/robot6axis/servo_4/servo_control/StatusStand AT 289 : BOOL := false;
    robot6axis_ctrled1/robot6axis/servo_4/servo_control/ActualPositionMa AT 6833 : REAL := 0.0;
    robot6axis_ctrled1/robot6axis/servo_4/servo_control/ActualVelocity AT 6834 : REAL := 0.0;
    robot6axis_ctrled1/robot6axis/servo_4/servo_control/MaximumVelocity AT 6835 : REAL := 0.0;
    robot6axis_ctrled1/robot6axis/servo_4/servo_control/VelEnabled AT 290 : BOOL := false;
    robot6axis_ctrled1/robot6axis/servo_4/servo_control/VelCmd AT 291 : BOOL := false;
    robot6axis_ctrled1/robot6axis/servo_4/servo_control/PosEnabled AT 292 : BOOL := false;
    robot6axis_ctrled1/robot6axis/servo_4/servo_control/PosCmd AT 293 : BOOL := false;
    robot6axis_ctrled1/robot6axis/servo_4/servo_control/Position AT 6837 : REAL := 0.0;
    robot6axis_ctrled1/robot6axis/servo_4/servo_control/Speed AT 6836 : REAL := 0.0;
    robot6axis_ctrled1/robot6axis/servo_4/servo_control/ManualMode AT 690 : INT := 0;
    robot6axis_ctrled1/robot6axis/servo_4/servo_control/initDone AT 297 : BOOL := false;
    robot6axis_ctrled1/robot6axis/servo_4/servo_control/ActualPositionMa1 AT 6847 : REAL := 0.0;
    robot6axis_ctrled1/robot6axis/servo_4/servo_control/offsetAxToMa1 AT 6848 : REAL := 0.0;
    robot6axis_ctrled1/robot6axis/servo_4/servo_control/HOME_POSITION AT 6849 : REAL := 100.0;
    robot6axis_ctrled1/robot6axis/servo_4/servo_control/MANUAL_POSITION1 AT 6850 : REAL := 0.0;
    robot6axis_ctrled1/robot6axis/servo_4/servo_control/MANUAL_POSITION2 AT 6851 : REAL := 150.0;
    robot6axis_ctrled1/robot6axis/servo_4/servo_control/MANUAL_SPEED1 AT 6852 : REAL := -100.0;
    robot6axis_ctrled1/robot6axis/servo_4/servo_control/MANUAL_SPEED2 AT 6853 : REAL := 100.0;
    robot6axis_ctrled1/robot6axis/servo_4/servo_control/MANUAL_SPEED AT 6854 : REAL := 100.0;
    robot6axis_ctrled1/robot6axis/servo_4/servo_velocity/MoveVelEnable AT 290 : BOOL := false;
    robot6axis_ctrled1/robot6axis/servo_4/servo_velocity/MoveVelStart AT 291 : BOOL := false;
    robot6axis_ctrled1/robot6axis/servo_4/servo_velocity/MoveSpeed AT 6836 : REAL := 0.0;
    robot6axis_ctrled1/robot6axis/servo_4/servo_velocity/MoveAcceleration AT 76 : REAL := 100.0;
    robot6axis_ctrled1/robot6axis/servo_4/servo_velocity/MoveDeceleration AT 75 : REAL := 100.0;
    robot6axis_ctrled1/robot6axis/servo_4/servo_velocity/MAX_SPEED AT 6469 : REAL(0.0..3.4e+038) := 30.0;
    robot6axis_ctrled1/robot6axis/servo_4/servo_velocity/MAX_ACCEL AT 6468 : REAL(0.0..3.4e+038) := 1500.0;
    robot6axis_ctrled1/robot6axis/servo_4/servo_velocity/MAX_DECEL AT 6467 : REAL(0.0..3.4e+038) := 1500.0;
    robot6axis_ctrled1/robot6axis/servo_4/servo_velocity/MODULO_LENGTH AT 6466 : REAL := 0.0;
    robot6axis_ctrled1/robot6axis/servo_4/servo_velocity/status AT 655 : INT := 0;
    robot6axis_ctrled1/robot6axis/servo_4/servo_velocity/errorFlag AT 654 : INT := 0;
    robot6axis_ctrled1/robot6axis/servo_4/servo_velocity/MoveVelDone AT 209 : BOOL := false;
    robot6axis_ctrled1/robot6axis/servo_4/servo_velocity/ActualPositionAx AT 6472 : REAL := 0.0;
    robot6axis_ctrled1/robot6axis/servo_4/servo_velocity/ActualVelocity AT 6471 : REAL := 0.0;
    robot6axis_ctrled1/robot6axis/servo_4/servo_velocity/firstStep AT 298 : BOOL := true;
    robot6axis_ctrled1/robot6axis/servo_4/servo_velocity/stepDone AT 299 : BOOL := false;
    robot6axis_ctrled1/robot6axis/servo_4/servo_velocity/currentTime AT 6855 : REAL := 0.0;
    robot6axis_ctrled1/robot6axis/servo_4/servo_velocity/MoveSpeed1 AT 6856 : REAL := 0.0;
    robot6axis_ctrled1/robot6axis/servo_4/servo_velocity/acceleration AT 6857 : REAL := 0.0;
    robot6axis_ctrled1/robot6axis/servo_4/servo_velocity/deceleration AT 6858 : REAL := 0.0;
    robot6axis_ctrled1/robot6axis/servo_4/servo_velocity/orderSpeed AT 6859 : REAL := 0.0;
    robot6axis_ctrled1/robot6axis/servo_4/servo_velocity/endChangeSpeed AT 6860 : REAL := 0.0;
    robot6axis_ctrled1/robot6axis/servo_4/servo_velocity/accelDecelChangeSpeed AT 6861 : REAL := 0.0;
    robot6axis_ctrled1/robot6axis/servo_4/servo_velocity/ActualVelocity1 AT 6862 : REAL := 0.0;
    robot6axis_ctrled1/robot6axis/servo_4/servo_velocity/speedChanged AT 300 : BOOL := false;
    robot6axis_ctrled1/robot6axis/servo_4/servo_position/MoveAbsEnable AT 292 : BOOL := false;
    robot6axis_ctrled1/robot6axis/servo_4/servo_position/MoveAbsStart AT 293 : BOOL := false;
    robot6axis_ctrled1/robot6axis/servo_4/servo_position/MovePosition AT 6837 : REAL := 0.0;
    robot6axis_ctrled1/robot6axis/servo_4/servo_position/MoveSpeed AT 6836 : REAL := 0.0;
    robot6axis_ctrled1/robot6axis/servo_4/servo_position/MoveAcceleration AT 76 : REAL := 100.0;
    robot6axis_ctrled1/robot6axis/servo_4/servo_position/MoveDeceleration AT 75 : REAL := 100.0;
    robot6axis_ctrled1/robot6axis/servo_4/servo_position/MAX_SPEED AT 6469 : REAL(0.0..3.4e+038) := 30.0;
    robot6axis_ctrled1/robot6axis/servo_4/servo_position/MAX_ACCEL AT 6468 : REAL(0.0..3.4e+038) := 1500.0;
    robot6axis_ctrled1/robot6axis/servo_4/servo_position/MAX_DECEL AT 6467 : REAL(0.0..3.4e+038) := 1500.0;
    robot6axis_ctrled1/robot6axis/servo_4/servo_position/MODULO_LENGTH AT 6466 : REAL := 0.0;
    robot6axis_ctrled1/robot6axis/servo_4/servo_position/status AT 655 : INT := 0;
    robot6axis_ctrled1/robot6axis/servo_4/servo_position/errorFlag AT 654 : INT := 0;
    robot6axis_ctrled1/robot6axis/servo_4/servo_position/MoveAbsDone AT 208 : BOOL := false;
    robot6axis_ctrled1/robot6axis/servo_4/servo_position/ActualPositionAx AT 6472 : REAL := 0.0;
    robot6axis_ctrled1/robot6axis/servo_4/servo_position/ActualVelocity AT 6471 : REAL := 0.0;
    robot6axis_ctrled1/robot6axis/servo_4/servo_position/firstStep AT 301 : BOOL := true;
    robot6axis_ctrled1/robot6axis/servo_4/servo_position/stepDone AT 302 : BOOL := false;
    robot6axis_ctrled1/robot6axis/servo_4/servo_position/timeToStop AT 6863 : REAL := 0.0;
    robot6axis_ctrled1/robot6axis/servo_4/servo_position/distanceToStop AT 6864 : REAL := 0.0;
    robot6axis_ctrled1/robot6axis/servo_4/servo_position/distance AT 6865 : REAL := 0.0;
    robot6axis_ctrled1/robot6axis/servo_4/servo_position/currentTime AT 6866 : REAL := 0.0;
    robot6axis_ctrled1/robot6axis/servo_4/servo_position/currentSpeed1 AT 6867 : REAL := 0.0;
    robot6axis_ctrled1/robot6axis/servo_4/servo_position/targetPosition AT 6868 : REAL := 0.0;
    robot6axis_ctrled1/robot6axis/servo_4/servo_position/ActualPositionAx1 AT 6869 : REAL := 0.0;
    robot6axis_ctrled1/robot6axis/servo_4/servo_position/acceleration AT 6870 : REAL := 0.0;
    robot6axis_ctrled1/robot6axis/servo_4/servo_position/deceleration AT 6871 : REAL := 0.0;
    robot6axis_ctrled1/robot6axis/servo_4/servo_position/orderSpeed AT 6872 : REAL := 0.0;
    robot6axis_ctrled1/robot6axis/servo_4/servo_position/moveDirection AT 6873 : REAL := 0.0;
    robot6axis_ctrled1/robot6axis/servo_4/servo_position/moveDirection1 AT 6874 : REAL := 0.0;
    robot6axis_ctrled1/robot6axis/servo_4/servo_position/endChangeSpeed AT 6875 : REAL := 0.0;
    robot6axis_ctrled1/robot6axis/servo_4/servo_position/ActualVelocity1 AT 6876 : REAL := 0.0;
    robot6axis_ctrled1/robot6axis/arm4/armOrigin AT 6564 : ARRAY[1..3] OF REAL := [3(0.0)];
    robot6axis_ctrled1/robot6axis/arm4/overallArmQuatInput AT 6569 : ARRAY[1..4] OF REAL := [4(0.0)];
    robot6axis_ctrled1/robot6axis/arm4/structRotVector AT 6458 : ARRAY[1..3] OF REAL := [2(0.0), 1.0];
    robot6axis_ctrled1/robot6axis/arm4/structRotDeg AT 6457 : REAL := 0.0;
    robot6axis_ctrled1/robot6axis/arm4/driveRotVector AT 128 : ARRAY[1..3] OF REAL := [1.0, 2(0.0)];
    robot6axis_ctrled1/robot6axis/arm4/driveRotDeg AT 6575 : REAL := 0.0;
    robot6axis_ctrled1/robot6axis/arm4/ownRotDeg AT 6456 : REAL := 0.0;
    robot6axis_ctrled1/robot6axis/arm4/driveResizeLength AT 6455 : REAL := 0.0;
    robot6axis_ctrled1/robot6axis/arm4/functionActive AT 202 : BOOL := false;
    robot6axis_ctrled1/robot6axis/arm4/armExtrem AT 6576 : ARRAY[1..3] OF REAL := [3(0.0)];
    robot6axis_ctrled1/robot6axis/arm4/overallArmRotOutput AT 6581 : ARRAY[1..4] OF REAL := [4(0.0)];
    robot6axis_ctrled1/robot6axis/arm4/productId AT 653 : DINT := -1;
    robot6axis_ctrled1/robot6axis/arm4/status_act_prod AT 691 : DINT := 0;
    robot6axis_ctrled1/robot6axis/arm4/m11 AT 6877 : REAL := 127.321;
    robot6axis_ctrled1/robot6axis/arm4/m12 AT 6878 : REAL := 0.0;
    robot6axis_ctrled1/robot6axis/arm4/m13 AT 6879 : REAL := 0.0;
    robot6axis_ctrled1/robot6axis/arm4/m14 AT 6880 : REAL := 453.404;
    robot6axis_ctrled1/robot6axis/arm4/m21 AT 6881 : REAL := 0.0;
    robot6axis_ctrled1/robot6axis/arm4/m22 AT 6882 : REAL := 1.0;
    robot6axis_ctrled1/robot6axis/arm4/m23 AT 6883 : REAL := 0.0;
    robot6axis_ctrled1/robot6axis/arm4/m24 AT 6884 : REAL := 1.0;
    robot6axis_ctrled1/robot6axis/arm4/m31 AT 6885 : REAL := 0.0;
    robot6axis_ctrled1/robot6axis/arm4/m32 AT 6886 : REAL := 0.0;
    robot6axis_ctrled1/robot6axis/arm4/m33 AT 6887 : REAL := 35.3669;
    robot6axis_ctrled1/robot6axis/arm4/m34 AT 6888 : REAL := 101.592;
    robot6axis_ctrled1/robot6axis/arm4/m41 AT 6889 : REAL := 0.0;
    robot6axis_ctrled1/robot6axis/arm4/m42 AT 6890 : REAL := 0.0;
    robot6axis_ctrled1/robot6axis/arm4/m43 AT 6891 : REAL := 0.0;
    robot6axis_ctrled1/robot6axis/arm4/m44 AT 6892 : REAL := 1.0;
    robot6axis_ctrled1/robot6axis/arm4/armLengthCalc AT 6893 : REAL := 0.0;
    robot6axis_ctrled1/robot6axis/arm4/functionActiveLocale AT 303 : BOOL := false;
    robot6axis_ctrled1/robot6axis/arm4/product_id AT 692 : DINT := -1;
    robot6axis_ctrled1/robot6axis/arm4/arm_id AT 693 : DINT := -1;
    robot6axis_ctrled1/robot6axis/arm4/timeToGripParam AT 6894 : REAL := 0.15;
    robot6axis_ctrled1/robot6axis/arm4/armLength AT 6895 : REAL := 202.0;
    robot6axis_ctrled1/robot6axis/arm4/armWidth AT 6896 : REAL := 40.0;
    robot6axis_ctrled1/robot6axis/arm4/armHeight AT 6897 : REAL := 40.0;
    robot6axis_ctrled1/robot6axis/arm4/armType AT 694 : INT := 0;
    robot6axis_ctrled1/robot6axis/servo_5/status AT 652 : INT := 0;
    robot6axis_ctrled1/robot6axis/servo_5/errorFlag AT 651 : INT := 0;
    robot6axis_ctrled1/robot6axis/servo_5/ActualPositionAx1 AT 6454 : REAL := 0.0;
    robot6axis_ctrled1/robot6axis/servo_5/MoveVelDone1 AT 201 : BOOL := false;
    robot6axis_ctrled1/robot6axis/servo_5/ActualVelocity1 AT 6453 : REAL := 0.0;
    robot6axis_ctrled1/robot6axis/servo_5/MoveAbsDone1 AT 200 : BOOL := false;
    robot6axis_ctrled1/robot6axis/servo_5/HomeCmd AT 70 : BOOL := false;
    robot6axis_ctrled1/robot6axis/servo_5/MoveVelCmd AT 69 : BOOL := false;
    robot6axis_ctrled1/robot6axis/servo_5/MoveAbsCmd AT 68 : BOOL := false;
    robot6axis_ctrled1/robot6axis/servo_5/MoveVel1ManualCmd AT 67 : BOOL := false;
    robot6axis_ctrled1/robot6axis/servo_5/MoveVel2ManualCmd AT 66 : BOOL := false;
    robot6axis_ctrled1/robot6axis/servo_5/MoveAbs1ManualCmd AT 65 : BOOL := false;
    robot6axis_ctrled1/robot6axis/servo_5/MoveAbs2ManualCmd AT 64 : BOOL := false;
    robot6axis_ctrled1/robot6axis/servo_5/StopCmd AT 22 : BOOL := false;
    robot6axis_ctrled1/robot6axis/servo_5/MovePosition AT 73 : REAL := 0.0;
    robot6axis_ctrled1/robot6axis/servo_5/MoveSpeed AT 72 : REAL := 100.0;
    robot6axis_ctrled1/robot6axis/servo_5/MoveAcceleration AT 71 : REAL := 100.0;
    robot6axis_ctrled1/robot6axis/servo_5/MoveDeceleration AT 70 : REAL := 100.0;
    robot6axis_ctrled1/robot6axis/servo_5/offsetAxToMa AT 69 : REAL := 0.0;
    robot6axis_ctrled1/robot6axis/servo_5/PLC_StatusReady AT 44 : BOOL := true;
    robot6axis_ctrled1/robot6axis/servo_5/PLC_StatusMoved AT 43 : BOOL := false;
    robot6axis_ctrled1/robot6axis/servo_5/PLC_StatusStand AT 42 : BOOL := false;
    robot6axis_ctrled1/robot6axis/servo_5/PLC_ActualPositionAx AT 171 : REAL := 0.0;
    robot6axis_ctrled1/robot6axis/servo_5/PLC_ActualPositionMa AT 55 : REAL := 0.0;
    robot6axis_ctrled1/robot6axis/servo_5/PLC_ActualVelocity AT 54 : REAL := 0.0;
    robot6axis_ctrled1/robot6axis/servo_5/physicalPosInit AT 6452 : REAL := 0.0;
    robot6axis_ctrled1/robot6axis/servo_5/MAX_SPEED AT 6451 : REAL(0.0..3.4e+038) := 30.0;
    robot6axis_ctrled1/robot6axis/servo_5/MAX_ACCEL AT 6450 : REAL(0.0..3.4e+038) := 1500.0;
    robot6axis_ctrled1/robot6axis/servo_5/MAX_DECEL AT 6449 : REAL(0.0..3.4e+038) := 1500.0;
    robot6axis_ctrled1/robot6axis/servo_5/MODULO_LENGTH AT 6448 : REAL := 0.0;
    robot6axis_ctrled1/robot6axis/servo_5/StatusReady AT 199 : BOOL := true;
    robot6axis_ctrled1/robot6axis/servo_5/StatusMoved AT 198 : BOOL := false;
    robot6axis_ctrled1/robot6axis/servo_5/StatusStand AT 197 : BOOL := false;
    robot6axis_ctrled1/robot6axis/servo_5/ActualPositionAx AT 6587 : REAL := 0.0;
    robot6axis_ctrled1/robot6axis/servo_5/ActualPositionMa AT 6447 : REAL := 0.0;
    robot6axis_ctrled1/robot6axis/servo_5/ActualVelocity AT 47 : REAL := 0.0;
    robot6axis_ctrled1/robot6axis/servo_5/MaximumVelocity AT 6446 : REAL := 0.0;
    robot6axis_ctrled1/robot6axis/servo_5/StatusPosIncrease AT 196 : BOOL := false;
    robot6axis_ctrled1/robot6axis/servo_5/StatusPosDecrease AT 195 : BOOL := false;
    robot6axis_ctrled1/robot6axis/servo_5/displayJauge AT 6445 : REAL := 0.0;
    robot6axis_ctrled1/robot6axis/servo_5/servo_mode/PLC_StatusReady AT 44 : BOOL := true;
    robot6axis_ctrled1/robot6axis/servo_5/servo_mode/PLC_StatusMoved AT 43 : BOOL := false;
    robot6axis_ctrled1/robot6axis/servo_5/servo_mode/PLC_StatusStand AT 42 : BOOL := false;
    robot6axis_ctrled1/robot6axis/servo_5/servo_mode/PLC_ActualPositionAx AT 171 : REAL := 0.0;
    robot6axis_ctrled1/robot6axis/servo_5/servo_mode/PLC_ActualPositionMa AT 55 : REAL := 0.0;
    robot6axis_ctrled1/robot6axis/servo_5/servo_mode/PLC_ActualVelocity AT 54 : REAL := 0.0;
    robot6axis_ctrled1/robot6axis/servo_5/servo_mode/StatusReady AT 304 : BOOL := true;
    robot6axis_ctrled1/robot6axis/servo_5/servo_mode/StatusMoved AT 305 : BOOL := false;
    robot6axis_ctrled1/robot6axis/servo_5/servo_mode/StatusStand AT 306 : BOOL := false;
    robot6axis_ctrled1/robot6axis/servo_5/servo_mode/ActualPositionMa AT 6898 : REAL := 0.0;
    robot6axis_ctrled1/robot6axis/servo_5/servo_mode/ActualVelocity AT 6899 : REAL := 0.0;
    robot6axis_ctrled1/robot6axis/servo_5/servo_mode/MaximumVelocity AT 6900 : REAL := 0.0;
    robot6axis_ctrled1/robot6axis/servo_5/servo_mode/physicalPosInit AT 6452 : REAL := 0.0;
    robot6axis_ctrled1/robot6axis/servo_5/servo_mode/ActualPositionAx AT 6454 : REAL := 0.0;
    robot6axis_ctrled1/robot6axis/servo_5/servo_mode/StatusReady_o AT 199 : BOOL := true;
    robot6axis_ctrled1/robot6axis/servo_5/servo_mode/StatusMoved_o AT 198 : BOOL := false;
    robot6axis_ctrled1/robot6axis/servo_5/servo_mode/StatusStand_o AT 197 : BOOL := false;
    robot6axis_ctrled1/robot6axis/servo_5/servo_mode/ActualPositionAx_o AT 6587 : REAL := 0.0;
    robot6axis_ctrled1/robot6axis/servo_5/servo_mode/ActualPositionMa_o AT 6447 : REAL := 0.0;
    robot6axis_ctrled1/robot6axis/servo_5/servo_mode/ActualVelocity_o AT 47 : REAL := 0.0;
    robot6axis_ctrled1/robot6axis/servo_5/servo_mode/MaximumVelocity_o AT 6446 : REAL := 0.0;
    robot6axis_ctrled1/robot6axis/servo_5/servo_mode/StatusPosIncrease_o AT 196 : BOOL := false;
    robot6axis_ctrled1/robot6axis/servo_5/servo_mode/StatusPosDecrease_o AT 195 : BOOL := false;
    robot6axis_ctrled1/robot6axis/servo_5/servo_mode/displayJauge_o AT 6445 : REAL := 0.0;
    robot6axis_ctrled1/robot6axis/servo_5/servo_mode/PLCMode AT 311 : BOOL := false;
    robot6axis_ctrled1/robot6axis/servo_5/servo_mode/PLCMode1 AT 312 : BOOL := false;
    robot6axis_ctrled1/robot6axis/servo_5/servo_mode/initDone AT 313 : BOOL := false;
    robot6axis_ctrled1/robot6axis/servo_5/servo_mode/displayPosMin AT 6903 : REAL := 0.0;
    robot6axis_ctrled1/robot6axis/servo_5/servo_mode/displayPosMax AT 6904 : REAL := 0.0;
    robot6axis_ctrled1/robot6axis/servo_5/servo_mode/PLC_ActualPositionAx1 AT 6905 : REAL := 0.0;
    robot6axis_ctrled1/robot6axis/servo_5/servo_mode/PLC_ActualVelocity1 AT 6906 : REAL := 0.0;
    robot6axis_ctrled1/robot6axis/servo_5/servo_mode/ActualPositionAx1 AT 6907 : REAL := 0.0;
    robot6axis_ctrled1/robot6axis/servo_5/servo_mode/ActualVelocity1 AT 6908 : REAL := 0.0;
    robot6axis_ctrled1/robot6axis/servo_5/servo_mode/offsetAxToMa AT 6909 : REAL := 0.0;
    robot6axis_ctrled1/robot6axis/servo_5/servo_mode/offsetAxToMa1 AT 6910 : REAL := 0.0;
    robot6axis_ctrled1/robot6axis/servo_5/servo_mode/ActualPositionMa_o1 AT 6911 : REAL := 0.0;
    robot6axis_ctrled1/robot6axis/servo_5/servo_control/HomeCmd AT 70 : BOOL := false;
    robot6axis_ctrled1/robot6axis/servo_5/servo_control/MoveVelCmd AT 69 : BOOL := false;
    robot6axis_ctrled1/robot6axis/servo_5/servo_control/MoveAbsCmd AT 68 : BOOL := false;
    robot6axis_ctrled1/robot6axis/servo_5/servo_control/MoveVel1ManualCmd AT 67 : BOOL := false;
    robot6axis_ctrled1/robot6axis/servo_5/servo_control/MoveVel2ManualCmd AT 66 : BOOL := false;
    robot6axis_ctrled1/robot6axis/servo_5/servo_control/MoveAbs1ManualCmd AT 65 : BOOL := false;
    robot6axis_ctrled1/robot6axis/servo_5/servo_control/MoveAbs2ManualCmd AT 64 : BOOL := false;
    robot6axis_ctrled1/robot6axis/servo_5/servo_control/StopCmd AT 22 : BOOL := false;
    robot6axis_ctrled1/robot6axis/servo_5/servo_control/MovePosition AT 73 : REAL := 0.0;
    robot6axis_ctrled1/robot6axis/servo_5/servo_control/MoveSpeed AT 72 : REAL := 100.0;
    robot6axis_ctrled1/robot6axis/servo_5/servo_control/MoveAcceleration AT 71 : REAL := 100.0;
    robot6axis_ctrled1/robot6axis/servo_5/servo_control/MoveDeceleration AT 70 : REAL := 100.0;
    robot6axis_ctrled1/robot6axis/servo_5/servo_control/offsetAxToMa AT 69 : REAL := 0.0;
    robot6axis_ctrled1/robot6axis/servo_5/servo_control/physicalPosInit AT 6452 : REAL := 0.0;
    robot6axis_ctrled1/robot6axis/servo_5/servo_control/MAX_SPEED AT 6451 : REAL(0.0..3.4e+038) := 30.0;
    robot6axis_ctrled1/robot6axis/servo_5/servo_control/status AT 652 : INT := 0;
    robot6axis_ctrled1/robot6axis/servo_5/servo_control/errorFlag AT 651 : INT := 0;
    robot6axis_ctrled1/robot6axis/servo_5/servo_control/IOActualPositionAx AT 6454 : REAL := 0.0;
    robot6axis_ctrled1/robot6axis/servo_5/servo_control/IOVelDone AT 201 : BOOL := false;
    robot6axis_ctrled1/robot6axis/servo_5/servo_control/IOAbsDone AT 200 : BOOL := false;
    robot6axis_ctrled1/robot6axis/servo_5/servo_control/IOActualVelocity AT 6453 : REAL := 0.0;
    robot6axis_ctrled1/robot6axis/servo_5/servo_control/OperationMode AT 695 : INT := 0;
    robot6axis_ctrled1/robot6axis/servo_5/servo_control/StatusReady AT 304 : BOOL := true;
    robot6axis_ctrled1/robot6axis/servo_5/servo_control/StatusMove AT 305 : BOOL := false;
    robot6axis_ctrled1/robot6axis/servo_5/servo_control/StatusStand AT 306 : BOOL := false;
    robot6axis_ctrled1/robot6axis/servo_5/servo_control/ActualPositionMa AT 6898 : REAL := 0.0;
    robot6axis_ctrled1/robot6axis/servo_5/servo_control/ActualVelocity AT 6899 : REAL := 0.0;
    robot6axis_ctrled1/robot6axis/servo_5/servo_control/MaximumVelocity AT 6900 : REAL := 0.0;
    robot6axis_ctrled1/robot6axis/servo_5/servo_control/VelEnabled AT 307 : BOOL := false;
    robot6axis_ctrled1/robot6axis/servo_5/servo_control/VelCmd AT 308 : BOOL := false;
    robot6axis_ctrled1/robot6axis/servo_5/servo_control/PosEnabled AT 309 : BOOL := false;
    robot6axis_ctrled1/robot6axis/servo_5/servo_control/PosCmd AT 310 : BOOL := false;
    robot6axis_ctrled1/robot6axis/servo_5/servo_control/Position AT 6902 : REAL := 0.0;
    robot6axis_ctrled1/robot6axis/servo_5/servo_control/Speed AT 6901 : REAL := 0.0;
    robot6axis_ctrled1/robot6axis/servo_5/servo_control/ManualMode AT 696 : INT := 0;
    robot6axis_ctrled1/robot6axis/servo_5/servo_control/initDone AT 314 : BOOL := false;
    robot6axis_ctrled1/robot6axis/servo_5/servo_control/ActualPositionMa1 AT 6912 : REAL := 0.0;
    robot6axis_ctrled1/robot6axis/servo_5/servo_control/offsetAxToMa1 AT 6913 : REAL := 0.0;
    robot6axis_ctrled1/robot6axis/servo_5/servo_control/HOME_POSITION AT 6914 : REAL := 100.0;
    robot6axis_ctrled1/robot6axis/servo_5/servo_control/MANUAL_POSITION1 AT 6915 : REAL := 0.0;
    robot6axis_ctrled1/robot6axis/servo_5/servo_control/MANUAL_POSITION2 AT 6916 : REAL := 150.0;
    robot6axis_ctrled1/robot6axis/servo_5/servo_control/MANUAL_SPEED1 AT 6917 : REAL := -100.0;
    robot6axis_ctrled1/robot6axis/servo_5/servo_control/MANUAL_SPEED2 AT 6918 : REAL := 100.0;
    robot6axis_ctrled1/robot6axis/servo_5/servo_control/MANUAL_SPEED AT 6919 : REAL := 100.0;
    robot6axis_ctrled1/robot6axis/servo_5/servo_velocity/MoveVelEnable AT 307 : BOOL := false;
    robot6axis_ctrled1/robot6axis/servo_5/servo_velocity/MoveVelStart AT 308 : BOOL := false;
    robot6axis_ctrled1/robot6axis/servo_5/servo_velocity/MoveSpeed AT 6901 : REAL := 0.0;
    robot6axis_ctrled1/robot6axis/servo_5/servo_velocity/MoveAcceleration AT 71 : REAL := 100.0;
    robot6axis_ctrled1/robot6axis/servo_5/servo_velocity/MoveDeceleration AT 70 : REAL := 100.0;
    robot6axis_ctrled1/robot6axis/servo_5/servo_velocity/MAX_SPEED AT 6451 : REAL(0.0..3.4e+038) := 30.0;
    robot6axis_ctrled1/robot6axis/servo_5/servo_velocity/MAX_ACCEL AT 6450 : REAL(0.0..3.4e+038) := 1500.0;
    robot6axis_ctrled1/robot6axis/servo_5/servo_velocity/MAX_DECEL AT 6449 : REAL(0.0..3.4e+038) := 1500.0;
    robot6axis_ctrled1/robot6axis/servo_5/servo_velocity/MODULO_LENGTH AT 6448 : REAL := 0.0;
    robot6axis_ctrled1/robot6axis/servo_5/servo_velocity/status AT 652 : INT := 0;
    robot6axis_ctrled1/robot6axis/servo_5/servo_velocity/errorFlag AT 651 : INT := 0;
    robot6axis_ctrled1/robot6axis/servo_5/servo_velocity/MoveVelDone AT 201 : BOOL := false;
    robot6axis_ctrled1/robot6axis/servo_5/servo_velocity/ActualPositionAx AT 6454 : REAL := 0.0;
    robot6axis_ctrled1/robot6axis/servo_5/servo_velocity/ActualVelocity AT 6453 : REAL := 0.0;
    robot6axis_ctrled1/robot6axis/servo_5/servo_velocity/firstStep AT 315 : BOOL := true;
    robot6axis_ctrled1/robot6axis/servo_5/servo_velocity/stepDone AT 316 : BOOL := false;
    robot6axis_ctrled1/robot6axis/servo_5/servo_velocity/currentTime AT 6920 : REAL := 0.0;
    robot6axis_ctrled1/robot6axis/servo_5/servo_velocity/MoveSpeed1 AT 6921 : REAL := 0.0;
    robot6axis_ctrled1/robot6axis/servo_5/servo_velocity/acceleration AT 6922 : REAL := 0.0;
    robot6axis_ctrled1/robot6axis/servo_5/servo_velocity/deceleration AT 6923 : REAL := 0.0;
    robot6axis_ctrled1/robot6axis/servo_5/servo_velocity/orderSpeed AT 6924 : REAL := 0.0;
    robot6axis_ctrled1/robot6axis/servo_5/servo_velocity/endChangeSpeed AT 6925 : REAL := 0.0;
    robot6axis_ctrled1/robot6axis/servo_5/servo_velocity/accelDecelChangeSpeed AT 6926 : REAL := 0.0;
    robot6axis_ctrled1/robot6axis/servo_5/servo_velocity/ActualVelocity1 AT 6927 : REAL := 0.0;
    robot6axis_ctrled1/robot6axis/servo_5/servo_velocity/speedChanged AT 317 : BOOL := false;
    robot6axis_ctrled1/robot6axis/servo_5/servo_position/MoveAbsEnable AT 309 : BOOL := false;
    robot6axis_ctrled1/robot6axis/servo_5/servo_position/MoveAbsStart AT 310 : BOOL := false;
    robot6axis_ctrled1/robot6axis/servo_5/servo_position/MovePosition AT 6902 : REAL := 0.0;
    robot6axis_ctrled1/robot6axis/servo_5/servo_position/MoveSpeed AT 6901 : REAL := 0.0;
    robot6axis_ctrled1/robot6axis/servo_5/servo_position/MoveAcceleration AT 71 : REAL := 100.0;
    robot6axis_ctrled1/robot6axis/servo_5/servo_position/MoveDeceleration AT 70 : REAL := 100.0;
    robot6axis_ctrled1/robot6axis/servo_5/servo_position/MAX_SPEED AT 6451 : REAL(0.0..3.4e+038) := 30.0;
    robot6axis_ctrled1/robot6axis/servo_5/servo_position/MAX_ACCEL AT 6450 : REAL(0.0..3.4e+038) := 1500.0;
    robot6axis_ctrled1/robot6axis/servo_5/servo_position/MAX_DECEL AT 6449 : REAL(0.0..3.4e+038) := 1500.0;
    robot6axis_ctrled1/robot6axis/servo_5/servo_position/MODULO_LENGTH AT 6448 : REAL := 0.0;
    robot6axis_ctrled1/robot6axis/servo_5/servo_position/status AT 652 : INT := 0;
    robot6axis_ctrled1/robot6axis/servo_5/servo_position/errorFlag AT 651 : INT := 0;
    robot6axis_ctrled1/robot6axis/servo_5/servo_position/MoveAbsDone AT 200 : BOOL := false;
    robot6axis_ctrled1/robot6axis/servo_5/servo_position/ActualPositionAx AT 6454 : REAL := 0.0;
    robot6axis_ctrled1/robot6axis/servo_5/servo_position/ActualVelocity AT 6453 : REAL := 0.0;
    robot6axis_ctrled1/robot6axis/servo_5/servo_position/firstStep AT 318 : BOOL := true;
    robot6axis_ctrled1/robot6axis/servo_5/servo_position/stepDone AT 319 : BOOL := false;
    robot6axis_ctrled1/robot6axis/servo_5/servo_position/timeToStop AT 6928 : REAL := 0.0;
    robot6axis_ctrled1/robot6axis/servo_5/servo_position/distanceToStop AT 6929 : REAL := 0.0;
    robot6axis_ctrled1/robot6axis/servo_5/servo_position/distance AT 6930 : REAL := 0.0;
    robot6axis_ctrled1/robot6axis/servo_5/servo_position/currentTime AT 6931 : REAL := 0.0;
    robot6axis_ctrled1/robot6axis/servo_5/servo_position/currentSpeed1 AT 6932 : REAL := 0.0;
    robot6axis_ctrled1/robot6axis/servo_5/servo_position/targetPosition AT 6933 : REAL := 0.0;
    robot6axis_ctrled1/robot6axis/servo_5/servo_position/ActualPositionAx1 AT 6934 : REAL := 0.0;
    robot6axis_ctrled1/robot6axis/servo_5/servo_position/acceleration AT 6935 : REAL := 0.0;
    robot6axis_ctrled1/robot6axis/servo_5/servo_position/deceleration AT 6936 : REAL := 0.0;
    robot6axis_ctrled1/robot6axis/servo_5/servo_position/orderSpeed AT 6937 : REAL := 0.0;
    robot6axis_ctrled1/robot6axis/servo_5/servo_position/moveDirection AT 6938 : REAL := 0.0;
    robot6axis_ctrled1/robot6axis/servo_5/servo_position/moveDirection1 AT 6939 : REAL := 0.0;
    robot6axis_ctrled1/robot6axis/servo_5/servo_position/endChangeSpeed AT 6940 : REAL := 0.0;
    robot6axis_ctrled1/robot6axis/servo_5/servo_position/ActualVelocity1 AT 6941 : REAL := 0.0;
    robot6axis_ctrled1/robot6axis/arm5/armOrigin AT 6576 : ARRAY[1..3] OF REAL := [3(0.0)];
    robot6axis_ctrled1/robot6axis/arm5/overallArmQuatInput AT 6581 : ARRAY[1..4] OF REAL := [4(0.0)];
    robot6axis_ctrled1/robot6axis/arm5/structRotVector AT 6440 : ARRAY[1..3] OF REAL := [2(0.0), 1.0];
    robot6axis_ctrled1/robot6axis/arm5/structRotDeg AT 6439 : REAL := 0.0;
    robot6axis_ctrled1/robot6axis/arm5/driveRotVector AT 123 : ARRAY[1..3] OF REAL := [0.0, 1.0, 0.0];
    robot6axis_ctrled1/robot6axis/arm5/driveRotDeg AT 6587 : REAL := 0.0;
    robot6axis_ctrled1/robot6axis/arm5/ownRotDeg AT 6438 : REAL := 0.0;
    robot6axis_ctrled1/robot6axis/arm5/driveResizeLength AT 6437 : REAL := 0.0;
    robot6axis_ctrled1/robot6axis/arm5/functionActive AT 194 : BOOL := false;
    robot6axis_ctrled1/robot6axis/arm5/armExtrem AT 6588 : ARRAY[1..3] OF REAL := [3(0.0)];
    robot6axis_ctrled1/robot6axis/arm5/overallArmRotOutput AT 6593 : ARRAY[1..4] OF REAL := [4(0.0)];
    robot6axis_ctrled1/robot6axis/arm5/productId AT 650 : DINT := -1;
    robot6axis_ctrled1/robot6axis/arm5/status_act_prod AT 697 : DINT := 0;
    robot6axis_ctrled1/robot6axis/arm5/m11 AT 6942 : REAL := 127.321;
    robot6axis_ctrled1/robot6axis/arm5/m12 AT 6943 : REAL := 0.0;
    robot6axis_ctrled1/robot6axis/arm5/m13 AT 6944 : REAL := 0.0;
    robot6axis_ctrled1/robot6axis/arm5/m14 AT 6945 : REAL := 453.404;
    robot6axis_ctrled1/robot6axis/arm5/m21 AT 6946 : REAL := 0.0;
    robot6axis_ctrled1/robot6axis/arm5/m22 AT 6947 : REAL := 1.0;
    robot6axis_ctrled1/robot6axis/arm5/m23 AT 6948 : REAL := 0.0;
    robot6axis_ctrled1/robot6axis/arm5/m24 AT 6949 : REAL := 1.0;
    robot6axis_ctrled1/robot6axis/arm5/m31 AT 6950 : REAL := 0.0;
    robot6axis_ctrled1/robot6axis/arm5/m32 AT 6951 : REAL := 0.0;
    robot6axis_ctrled1/robot6axis/arm5/m33 AT 6952 : REAL := 35.3669;
    robot6axis_ctrled1/robot6axis/arm5/m34 AT 6953 : REAL := 46.0654;
    robot6axis_ctrled1/robot6axis/arm5/m41 AT 6954 : REAL := 0.0;
    robot6axis_ctrled1/robot6axis/arm5/m42 AT 6955 : REAL := 0.0;
    robot6axis_ctrled1/robot6axis/arm5/m43 AT 6956 : REAL := 0.0;
    robot6axis_ctrled1/robot6axis/arm5/m44 AT 6957 : REAL := 1.0;
    robot6axis_ctrled1/robot6axis/arm5/armLengthCalc AT 6958 : REAL := 0.0;
    robot6axis_ctrled1/robot6axis/arm5/functionActiveLocale AT 320 : BOOL := false;
    robot6axis_ctrled1/robot6axis/arm5/product_id AT 698 : DINT := -1;
    robot6axis_ctrled1/robot6axis/arm5/arm_id AT 699 : DINT := -1;
    robot6axis_ctrled1/robot6axis/arm5/timeToGripParam AT 6959 : REAL := 0.15;
    robot6axis_ctrled1/robot6axis/arm5/armLength AT 6960 : REAL := 61.0;
    robot6axis_ctrled1/robot6axis/arm5/armWidth AT 6961 : REAL := 40.0;
    robot6axis_ctrled1/robot6axis/arm5/armHeight AT 6962 : REAL := 40.0;
    robot6axis_ctrled1/robot6axis/arm5/armType AT 700 : INT := 0;
    robot6axis_ctrled1/robot6axis/servo_6/status AT 649 : INT := 0;
    robot6axis_ctrled1/robot6axis/servo_6/errorFlag AT 648 : INT := 0;
    robot6axis_ctrled1/robot6axis/servo_6/ActualPositionAx1 AT 6436 : REAL := 0.0;
    robot6axis_ctrled1/robot6axis/servo_6/MoveVelDone1 AT 193 : BOOL := false;
    robot6axis_ctrled1/robot6axis/servo_6/ActualVelocity1 AT 6435 : REAL := 0.0;
    robot6axis_ctrled1/robot6axis/servo_6/MoveAbsDone1 AT 192 : BOOL := false;
    robot6axis_ctrled1/robot6axis/servo_6/HomeCmd AT 63 : BOOL := false;
    robot6axis_ctrled1/robot6axis/servo_6/MoveVelCmd AT 62 : BOOL := false;
    robot6axis_ctrled1/robot6axis/servo_6/MoveAbsCmd AT 61 : BOOL := false;
    robot6axis_ctrled1/robot6axis/servo_6/MoveVel1ManualCmd AT 60 : BOOL := false;
    robot6axis_ctrled1/robot6axis/servo_6/MoveVel2ManualCmd AT 59 : BOOL := false;
    robot6axis_ctrled1/robot6axis/servo_6/MoveAbs1ManualCmd AT 58 : BOOL := false;
    robot6axis_ctrled1/robot6axis/servo_6/MoveAbs2ManualCmd AT 57 : BOOL := false;
    robot6axis_ctrled1/robot6axis/servo_6/StopCmd AT 22 : BOOL := false;
    robot6axis_ctrled1/robot6axis/servo_6/MovePosition AT 68 : REAL := 0.0;
    robot6axis_ctrled1/robot6axis/servo_6/MoveSpeed AT 67 : REAL := 100.0;
    robot6axis_ctrled1/robot6axis/servo_6/MoveAcceleration AT 66 : REAL := 100.0;
    robot6axis_ctrled1/robot6axis/servo_6/MoveDeceleration AT 65 : REAL := 100.0;
    robot6axis_ctrled1/robot6axis/servo_6/offsetAxToMa AT 64 : REAL := 0.0;
    robot6axis_ctrled1/robot6axis/servo_6/PLC_StatusReady AT 41 : BOOL := true;
    robot6axis_ctrled1/robot6axis/servo_6/PLC_StatusMoved AT 40 : BOOL := false;
    robot6axis_ctrled1/robot6axis/servo_6/PLC_StatusStand AT 39 : BOOL := false;
    robot6axis_ctrled1/robot6axis/servo_6/PLC_ActualPositionAx AT 172 : REAL := 0.0;
    robot6axis_ctrled1/robot6axis/servo_6/PLC_ActualPositionMa AT 53 : REAL := 0.0;
    robot6axis_ctrled1/robot6axis/servo_6/PLC_ActualVelocity AT 52 : REAL := 0.0;
    robot6axis_ctrled1/robot6axis/servo_6/physicalPosInit AT 6434 : REAL := 0.0;
    robot6axis_ctrled1/robot6axis/servo_6/MAX_SPEED AT 6433 : REAL(0.0..3.4e+038) := 30.0;
    robot6axis_ctrled1/robot6axis/servo_6/MAX_ACCEL AT 6432 : REAL(0.0..3.4e+038) := 1500.0;
    robot6axis_ctrled1/robot6axis/servo_6/MAX_DECEL AT 6431 : REAL(0.0..3.4e+038) := 1500.0;
    robot6axis_ctrled1/robot6axis/servo_6/MODULO_LENGTH AT 6430 : REAL := 0.0;
    robot6axis_ctrled1/robot6axis/servo_6/StatusReady AT 191 : BOOL := true;
    robot6axis_ctrled1/robot6axis/servo_6/StatusMoved AT 190 : BOOL := false;
    robot6axis_ctrled1/robot6axis/servo_6/StatusStand AT 189 : BOOL := false;
    robot6axis_ctrled1/robot6axis/servo_6/ActualPositionAx AT 6599 : REAL := 0.0;
    robot6axis_ctrled1/robot6axis/servo_6/ActualPositionMa AT 6429 : REAL := 0.0;
    robot6axis_ctrled1/robot6axis/servo_6/ActualVelocity AT 46 : REAL := 0.0;
    robot6axis_ctrled1/robot6axis/servo_6/MaximumVelocity AT 6428 : REAL := 0.0;
    robot6axis_ctrled1/robot6axis/servo_6/StatusPosIncrease AT 188 : BOOL := false;
    robot6axis_ctrled1/robot6axis/servo_6/StatusPosDecrease AT 187 : BOOL := false;
    robot6axis_ctrled1/robot6axis/servo_6/displayJauge AT 6427 : REAL := 0.0;
    robot6axis_ctrled1/robot6axis/servo_6/servo_mode/PLC_StatusReady AT 41 : BOOL := true;
    robot6axis_ctrled1/robot6axis/servo_6/servo_mode/PLC_StatusMoved AT 40 : BOOL := false;
    robot6axis_ctrled1/robot6axis/servo_6/servo_mode/PLC_StatusStand AT 39 : BOOL := false;
    robot6axis_ctrled1/robot6axis/servo_6/servo_mode/PLC_ActualPositionAx AT 172 : REAL := 0.0;
    robot6axis_ctrled1/robot6axis/servo_6/servo_mode/PLC_ActualPositionMa AT 53 : REAL := 0.0;
    robot6axis_ctrled1/robot6axis/servo_6/servo_mode/PLC_ActualVelocity AT 52 : REAL := 0.0;
    robot6axis_ctrled1/robot6axis/servo_6/servo_mode/StatusReady AT 321 : BOOL := true;
    robot6axis_ctrled1/robot6axis/servo_6/servo_mode/StatusMoved AT 322 : BOOL := false;
    robot6axis_ctrled1/robot6axis/servo_6/servo_mode/StatusStand AT 323 : BOOL := false;
    robot6axis_ctrled1/robot6axis/servo_6/servo_mode/ActualPositionMa AT 6963 : REAL := 0.0;
    robot6axis_ctrled1/robot6axis/servo_6/servo_mode/ActualVelocity AT 6964 : REAL := 0.0;
    robot6axis_ctrled1/robot6axis/servo_6/servo_mode/MaximumVelocity AT 6965 : REAL := 0.0;
    robot6axis_ctrled1/robot6axis/servo_6/servo_mode/physicalPosInit AT 6434 : REAL := 0.0;
    robot6axis_ctrled1/robot6axis/servo_6/servo_mode/ActualPositionAx AT 6436 : REAL := 0.0;
    robot6axis_ctrled1/robot6axis/servo_6/servo_mode/StatusReady_o AT 191 : BOOL := true;
    robot6axis_ctrled1/robot6axis/servo_6/servo_mode/StatusMoved_o AT 190 : BOOL := false;
    robot6axis_ctrled1/robot6axis/servo_6/servo_mode/StatusStand_o AT 189 : BOOL := false;
    robot6axis_ctrled1/robot6axis/servo_6/servo_mode/ActualPositionAx_o AT 6599 : REAL := 0.0;
    robot6axis_ctrled1/robot6axis/servo_6/servo_mode/ActualPositionMa_o AT 6429 : REAL := 0.0;
    robot6axis_ctrled1/robot6axis/servo_6/servo_mode/ActualVelocity_o AT 46 : REAL := 0.0;
    robot6axis_ctrled1/robot6axis/servo_6/servo_mode/MaximumVelocity_o AT 6428 : REAL := 0.0;
    robot6axis_ctrled1/robot6axis/servo_6/servo_mode/StatusPosIncrease_o AT 188 : BOOL := false;
    robot6axis_ctrled1/robot6axis/servo_6/servo_mode/StatusPosDecrease_o AT 187 : BOOL := false;
    robot6axis_ctrled1/robot6axis/servo_6/servo_mode/displayJauge_o AT 6427 : REAL := 0.0;
    robot6axis_ctrled1/robot6axis/servo_6/servo_mode/PLCMode AT 328 : BOOL := false;
    robot6axis_ctrled1/robot6axis/servo_6/servo_mode/PLCMode1 AT 329 : BOOL := false;
    robot6axis_ctrled1/robot6axis/servo_6/servo_mode/initDone AT 330 : BOOL := false;
    robot6axis_ctrled1/robot6axis/servo_6/servo_mode/displayPosMin AT 6968 : REAL := 0.0;
    robot6axis_ctrled1/robot6axis/servo_6/servo_mode/displayPosMax AT 6969 : REAL := 0.0;
    robot6axis_ctrled1/robot6axis/servo_6/servo_mode/PLC_ActualPositionAx1 AT 6970 : REAL := 0.0;
    robot6axis_ctrled1/robot6axis/servo_6/servo_mode/PLC_ActualVelocity1 AT 6971 : REAL := 0.0;
    robot6axis_ctrled1/robot6axis/servo_6/servo_mode/ActualPositionAx1 AT 6972 : REAL := 0.0;
    robot6axis_ctrled1/robot6axis/servo_6/servo_mode/ActualVelocity1 AT 6973 : REAL := 0.0;
    robot6axis_ctrled1/robot6axis/servo_6/servo_mode/offsetAxToMa AT 6974 : REAL := 0.0;
    robot6axis_ctrled1/robot6axis/servo_6/servo_mode/offsetAxToMa1 AT 6975 : REAL := 0.0;
    robot6axis_ctrled1/robot6axis/servo_6/servo_mode/ActualPositionMa_o1 AT 6976 : REAL := 0.0;
    robot6axis_ctrled1/robot6axis/servo_6/servo_control/HomeCmd AT 63 : BOOL := false;
    robot6axis_ctrled1/robot6axis/servo_6/servo_control/MoveVelCmd AT 62 : BOOL := false;
    robot6axis_ctrled1/robot6axis/servo_6/servo_control/MoveAbsCmd AT 61 : BOOL := false;
    robot6axis_ctrled1/robot6axis/servo_6/servo_control/MoveVel1ManualCmd AT 60 : BOOL := false;
    robot6axis_ctrled1/robot6axis/servo_6/servo_control/MoveVel2ManualCmd AT 59 : BOOL := false;
    robot6axis_ctrled1/robot6axis/servo_6/servo_control/MoveAbs1ManualCmd AT 58 : BOOL := false;
    robot6axis_ctrled1/robot6axis/servo_6/servo_control/MoveAbs2ManualCmd AT 57 : BOOL := false;
    robot6axis_ctrled1/robot6axis/servo_6/servo_control/StopCmd AT 22 : BOOL := false;
    robot6axis_ctrled1/robot6axis/servo_6/servo_control/MovePosition AT 68 : REAL := 0.0;
    robot6axis_ctrled1/robot6axis/servo_6/servo_control/MoveSpeed AT 67 : REAL := 100.0;
    robot6axis_ctrled1/robot6axis/servo_6/servo_control/MoveAcceleration AT 66 : REAL := 100.0;
    robot6axis_ctrled1/robot6axis/servo_6/servo_control/MoveDeceleration AT 65 : REAL := 100.0;
    robot6axis_ctrled1/robot6axis/servo_6/servo_control/offsetAxToMa AT 64 : REAL := 0.0;
    robot6axis_ctrled1/robot6axis/servo_6/servo_control/physicalPosInit AT 6434 : REAL := 0.0;
    robot6axis_ctrled1/robot6axis/servo_6/servo_control/MAX_SPEED AT 6433 : REAL(0.0..3.4e+038) := 30.0;
    robot6axis_ctrled1/robot6axis/servo_6/servo_control/status AT 649 : INT := 0;
    robot6axis_ctrled1/robot6axis/servo_6/servo_control/errorFlag AT 648 : INT := 0;
    robot6axis_ctrled1/robot6axis/servo_6/servo_control/IOActualPositionAx AT 6436 : REAL := 0.0;
    robot6axis_ctrled1/robot6axis/servo_6/servo_control/IOVelDone AT 193 : BOOL := false;
    robot6axis_ctrled1/robot6axis/servo_6/servo_control/IOAbsDone AT 192 : BOOL := false;
    robot6axis_ctrled1/robot6axis/servo_6/servo_control/IOActualVelocity AT 6435 : REAL := 0.0;
    robot6axis_ctrled1/robot6axis/servo_6/servo_control/OperationMode AT 701 : INT := 0;
    robot6axis_ctrled1/robot6axis/servo_6/servo_control/StatusReady AT 321 : BOOL := true;
    robot6axis_ctrled1/robot6axis/servo_6/servo_control/StatusMove AT 322 : BOOL := false;
    robot6axis_ctrled1/robot6axis/servo_6/servo_control/StatusStand AT 323 : BOOL := false;
    robot6axis_ctrled1/robot6axis/servo_6/servo_control/ActualPositionMa AT 6963 : REAL := 0.0;
    robot6axis_ctrled1/robot6axis/servo_6/servo_control/ActualVelocity AT 6964 : REAL := 0.0;
    robot6axis_ctrled1/robot6axis/servo_6/servo_control/MaximumVelocity AT 6965 : REAL := 0.0;
    robot6axis_ctrled1/robot6axis/servo_6/servo_control/VelEnabled AT 324 : BOOL := false;
    robot6axis_ctrled1/robot6axis/servo_6/servo_control/VelCmd AT 325 : BOOL := false;
    robot6axis_ctrled1/robot6axis/servo_6/servo_control/PosEnabled AT 326 : BOOL := false;
    robot6axis_ctrled1/robot6axis/servo_6/servo_control/PosCmd AT 327 : BOOL := false;
    robot6axis_ctrled1/robot6axis/servo_6/servo_control/Position AT 6967 : REAL := 0.0;
    robot6axis_ctrled1/robot6axis/servo_6/servo_control/Speed AT 6966 : REAL := 0.0;
    robot6axis_ctrled1/robot6axis/servo_6/servo_control/ManualMode AT 702 : INT := 0;
    robot6axis_ctrled1/robot6axis/servo_6/servo_control/initDone AT 331 : BOOL := false;
    robot6axis_ctrled1/robot6axis/servo_6/servo_control/ActualPositionMa1 AT 6977 : REAL := 0.0;
    robot6axis_ctrled1/robot6axis/servo_6/servo_control/offsetAxToMa1 AT 6978 : REAL := 0.0;
    robot6axis_ctrled1/robot6axis/servo_6/servo_control/HOME_POSITION AT 6979 : REAL := 100.0;
    robot6axis_ctrled1/robot6axis/servo_6/servo_control/MANUAL_POSITION1 AT 6980 : REAL := 0.0;
    robot6axis_ctrled1/robot6axis/servo_6/servo_control/MANUAL_POSITION2 AT 6981 : REAL := 150.0;
    robot6axis_ctrled1/robot6axis/servo_6/servo_control/MANUAL_SPEED1 AT 6982 : REAL := -100.0;
    robot6axis_ctrled1/robot6axis/servo_6/servo_control/MANUAL_SPEED2 AT 6983 : REAL := 100.0;
    robot6axis_ctrled1/robot6axis/servo_6/servo_control/MANUAL_SPEED AT 6984 : REAL := 100.0;
    robot6axis_ctrled1/robot6axis/servo_6/servo_velocity/MoveVelEnable AT 324 : BOOL := false;
    robot6axis_ctrled1/robot6axis/servo_6/servo_velocity/MoveVelStart AT 325 : BOOL := false;
    robot6axis_ctrled1/robot6axis/servo_6/servo_velocity/MoveSpeed AT 6966 : REAL := 0.0;
    robot6axis_ctrled1/robot6axis/servo_6/servo_velocity/MoveAcceleration AT 66 : REAL := 100.0;
    robot6axis_ctrled1/robot6axis/servo_6/servo_velocity/MoveDeceleration AT 65 : REAL := 100.0;
    robot6axis_ctrled1/robot6axis/servo_6/servo_velocity/MAX_SPEED AT 6433 : REAL(0.0..3.4e+038) := 30.0;
    robot6axis_ctrled1/robot6axis/servo_6/servo_velocity/MAX_ACCEL AT 6432 : REAL(0.0..3.4e+038) := 1500.0;
    robot6axis_ctrled1/robot6axis/servo_6/servo_velocity/MAX_DECEL AT 6431 : REAL(0.0..3.4e+038) := 1500.0;
    robot6axis_ctrled1/robot6axis/servo_6/servo_velocity/MODULO_LENGTH AT 6430 : REAL := 0.0;
    robot6axis_ctrled1/robot6axis/servo_6/servo_velocity/status AT 649 : INT := 0;
    robot6axis_ctrled1/robot6axis/servo_6/servo_velocity/errorFlag AT 648 : INT := 0;
    robot6axis_ctrled1/robot6axis/servo_6/servo_velocity/MoveVelDone AT 193 : BOOL := false;
    robot6axis_ctrled1/robot6axis/servo_6/servo_velocity/ActualPositionAx AT 6436 : REAL := 0.0;
    robot6axis_ctrled1/robot6axis/servo_6/servo_velocity/ActualVelocity AT 6435 : REAL := 0.0;
    robot6axis_ctrled1/robot6axis/servo_6/servo_velocity/firstStep AT 332 : BOOL := true;
    robot6axis_ctrled1/robot6axis/servo_6/servo_velocity/stepDone AT 333 : BOOL := false;
    robot6axis_ctrled1/robot6axis/servo_6/servo_velocity/currentTime AT 6985 : REAL := 0.0;
    robot6axis_ctrled1/robot6axis/servo_6/servo_velocity/MoveSpeed1 AT 6986 : REAL := 0.0;
    robot6axis_ctrled1/robot6axis/servo_6/servo_velocity/acceleration AT 6987 : REAL := 0.0;
    robot6axis_ctrled1/robot6axis/servo_6/servo_velocity/deceleration AT 6988 : REAL := 0.0;
    robot6axis_ctrled1/robot6axis/servo_6/servo_velocity/orderSpeed AT 6989 : REAL := 0.0;
    robot6axis_ctrled1/robot6axis/servo_6/servo_velocity/endChangeSpeed AT 6990 : REAL := 0.0;
    robot6axis_ctrled1/robot6axis/servo_6/servo_velocity/accelDecelChangeSpeed AT 6991 : REAL := 0.0;
    robot6axis_ctrled1/robot6axis/servo_6/servo_velocity/ActualVelocity1 AT 6992 : REAL := 0.0;
    robot6axis_ctrled1/robot6axis/servo_6/servo_velocity/speedChanged AT 334 : BOOL := false;
    robot6axis_ctrled1/robot6axis/servo_6/servo_position/MoveAbsEnable AT 326 : BOOL := false;
    robot6axis_ctrled1/robot6axis/servo_6/servo_position/MoveAbsStart AT 327 : BOOL := false;
    robot6axis_ctrled1/robot6axis/servo_6/servo_position/MovePosition AT 6967 : REAL := 0.0;
    robot6axis_ctrled1/robot6axis/servo_6/servo_position/MoveSpeed AT 6966 : REAL := 0.0;
    robot6axis_ctrled1/robot6axis/servo_6/servo_position/MoveAcceleration AT 66 : REAL := 100.0;
    robot6axis_ctrled1/robot6axis/servo_6/servo_position/MoveDeceleration AT 65 : REAL := 100.0;
    robot6axis_ctrled1/robot6axis/servo_6/servo_position/MAX_SPEED AT 6433 : REAL(0.0..3.4e+038) := 30.0;
    robot6axis_ctrled1/robot6axis/servo_6/servo_position/MAX_ACCEL AT 6432 : REAL(0.0..3.4e+038) := 1500.0;
    robot6axis_ctrled1/robot6axis/servo_6/servo_position/MAX_DECEL AT 6431 : REAL(0.0..3.4e+038) := 1500.0;
    robot6axis_ctrled1/robot6axis/servo_6/servo_position/MODULO_LENGTH AT 6430 : REAL := 0.0;
    robot6axis_ctrled1/robot6axis/servo_6/servo_position/status AT 649 : INT := 0;
    robot6axis_ctrled1/robot6axis/servo_6/servo_position/errorFlag AT 648 : INT := 0;
    robot6axis_ctrled1/robot6axis/servo_6/servo_position/MoveAbsDone AT 192 : BOOL := false;
    robot6axis_ctrled1/robot6axis/servo_6/servo_position/ActualPositionAx AT 6436 : REAL := 0.0;
    robot6axis_ctrled1/robot6axis/servo_6/servo_position/ActualVelocity AT 6435 : REAL := 0.0;
    robot6axis_ctrled1/robot6axis/servo_6/servo_position/firstStep AT 335 : BOOL := true;
    robot6axis_ctrled1/robot6axis/servo_6/servo_position/stepDone AT 336 : BOOL := false;
    robot6axis_ctrled1/robot6axis/servo_6/servo_position/timeToStop AT 6993 : REAL := 0.0;
    robot6axis_ctrled1/robot6axis/servo_6/servo_position/distanceToStop AT 6994 : REAL := 0.0;
    robot6axis_ctrled1/robot6axis/servo_6/servo_position/distance AT 6995 : REAL := 0.0;
    robot6axis_ctrled1/robot6axis/servo_6/servo_position/currentTime AT 6996 : REAL := 0.0;
    robot6axis_ctrled1/robot6axis/servo_6/servo_position/currentSpeed1 AT 6997 : REAL := 0.0;
    robot6axis_ctrled1/robot6axis/servo_6/servo_position/targetPosition AT 6998 : REAL := 0.0;
    robot6axis_ctrled1/robot6axis/servo_6/servo_position/ActualPositionAx1 AT 6999 : REAL := 0.0;
    robot6axis_ctrled1/robot6axis/servo_6/servo_position/acceleration AT 7000 : REAL := 0.0;
    robot6axis_ctrled1/robot6axis/servo_6/servo_position/deceleration AT 7001 : REAL := 0.0;
    robot6axis_ctrled1/robot6axis/servo_6/servo_position/orderSpeed AT 7002 : REAL := 0.0;
    robot6axis_ctrled1/robot6axis/servo_6/servo_position/moveDirection AT 7003 : REAL := 0.0;
    robot6axis_ctrled1/robot6axis/servo_6/servo_position/moveDirection1 AT 7004 : REAL := 0.0;
    robot6axis_ctrled1/robot6axis/servo_6/servo_position/endChangeSpeed AT 7005 : REAL := 0.0;
    robot6axis_ctrled1/robot6axis/servo_6/servo_position/ActualVelocity1 AT 7006 : REAL := 0.0;
    robot6axis_ctrled1/robot6axis/arm6/armOrigin AT 6588 : ARRAY[1..3] OF REAL := [3(0.0)];
    robot6axis_ctrled1/robot6axis/arm6/overallArmQuatInput AT 6593 : ARRAY[1..4] OF REAL := [4(0.0)];
    robot6axis_ctrled1/robot6axis/arm6/structRotVector AT 6422 : ARRAY[1..3] OF REAL := [2(0.0), 1.0];
    robot6axis_ctrled1/robot6axis/arm6/structRotDeg AT 6421 : REAL := 0.0;
    robot6axis_ctrled1/robot6axis/arm6/driveRotVector AT 118 : ARRAY[1..3] OF REAL := [1.0, 2(0.0)];
    robot6axis_ctrled1/robot6axis/arm6/driveRotDeg AT 6599 : REAL := 0.0;
    robot6axis_ctrled1/robot6axis/arm6/ownRotDeg AT 6420 : REAL := 0.0;
    robot6axis_ctrled1/robot6axis/arm6/driveResizeLength AT 6419 : REAL := 0.0;
    robot6axis_ctrled1/robot6axis/arm6/functionActive AT 186 : BOOL := false;
    robot6axis_ctrled1/robot6axis/arm6/armExtrem AT 22 : ARRAY[1..3] OF REAL := [3(0.0)];
    robot6axis_ctrled1/robot6axis/arm6/overallArmRotOutput AT 6600 : ARRAY[1..4] OF REAL := [4(0.0)];
    robot6axis_ctrled1/robot6axis/arm6/productId AT 666 : DINT := -1;
    robot6axis_ctrled1/robot6axis/arm6/status_act_prod AT 703 : DINT := 0;
    robot6axis_ctrled1/robot6axis/arm6/m11 AT 7007 : REAL := 128.028;
    robot6axis_ctrled1/robot6axis/arm6/m12 AT 7008 : REAL := 0.0;
    robot6axis_ctrled1/robot6axis/arm6/m13 AT 7009 : REAL := 0.0;
    robot6axis_ctrled1/robot6axis/arm6/m14 AT 7010 : REAL := 459.77;
    robot6axis_ctrled1/robot6axis/arm6/m21 AT 7011 : REAL := 0.0;
    robot6axis_ctrled1/robot6axis/arm6/m22 AT 7012 : REAL := 1.0;
    robot6axis_ctrled1/robot6axis/arm6/m23 AT 7013 : REAL := 0.0;
    robot6axis_ctrled1/robot6axis/arm6/m24 AT 7014 : REAL := 1.0;
    robot6axis_ctrled1/robot6axis/arm6/m31 AT 7015 : REAL := 0.0;
    robot6axis_ctrled1/robot6axis/arm6/m32 AT 7016 : REAL := 0.0;
    robot6axis_ctrled1/robot6axis/arm6/m33 AT 7017 : REAL := 35.3669;
    robot6axis_ctrled1/robot6axis/arm6/m34 AT 7018 : REAL := -10.5217;
    robot6axis_ctrled1/robot6axis/arm6/m41 AT 7019 : REAL := 0.0;
    robot6axis_ctrled1/robot6axis/arm6/m42 AT 7020 : REAL := 0.0;
    robot6axis_ctrled1/robot6axis/arm6/m43 AT 7021 : REAL := 0.0;
    robot6axis_ctrled1/robot6axis/arm6/m44 AT 7022 : REAL := 1.0;
    robot6axis_ctrled1/robot6axis/arm6/armLengthCalc AT 7023 : REAL := 0.0;
    robot6axis_ctrled1/robot6axis/arm6/functionActiveLocale AT 337 : BOOL := false;
    robot6axis_ctrled1/robot6axis/arm6/product_id AT 704 : DINT := -1;
    robot6axis_ctrled1/robot6axis/arm6/arm_id AT 705 : DINT := -1;
    robot6axis_ctrled1/robot6axis/arm6/timeToGripParam AT 7024 : REAL := 0.15;
    robot6axis_ctrled1/robot6axis/arm6/armLength AT 7025 : REAL := 9.0;
    robot6axis_ctrled1/robot6axis/arm6/armWidth AT 7026 : REAL := 5.0;
    robot6axis_ctrled1/robot6axis/arm6/armHeight AT 7027 : REAL := 5.0;
    robot6axis_ctrled1/robot6axis/arm6/armType AT 706 : INT := 0;
    robot6axis_ctrled1/robot6axis/function_trigger/armExtrem AT 22 : ARRAY[1..3] OF REAL := [3(0.0)];
    robot6axis_ctrled1/robot6axis/function_trigger/productId AT 666 : DINT := -1;
    robot6axis_ctrled1/robot6axis/function_trigger/velX AT 21 : REAL := 0.0;
    robot6axis_ctrled1/robot6axis/function_trigger/velY AT 20 : REAL := 0.0;
    robot6axis_ctrled1/robot6axis/function_trigger/velZ AT 19 : REAL := 0.0;
    robot6axis_ctrled1/robot6axis/function_trigger/armInStop AT 5 : BOOL := false;
    robot6axis_ctrled1/robot6axis/function_trigger/armExtrem1 AT 7028 : ARRAY[1..3] OF REAL := [3(0.0)];
    robot6axis_ctrled1/robot6axis/function_trigger/i AT 707 : INT := 0;
    robot6axis_ctrled1/robot6axis/function_trigger/productTimeDetect AT 7033 : REAL := 0.0;
    robot6axis_ctrled1/robot6axis/function_trigger/productDetected AT 338 : BOOL := false;
    robot6axis_ctrled1/robot6axis/function_trigger/productId1 AT 708 : DINT := -1;
    robot6axis_ctrled1/robot6axis/function_trigger/actionTake AT 339 : BOOL := false;
    robot6axis_ctrled1/robot6axis/function_trigger/activeArea AT 340 : BOOL := false;
    robot6axis_ctrled1/robot6axis/function_trigger/ACTIVE_AREA_Z AT 7034 : REAL := 1100.0;
    robot6axis_ctrled1/robot6axis/function_trigger/TEMPO_DETECTION_PRO AT 7035 : REAL := 0.2;
    robot6axis_ctrled1/robot6axis/arm1RowA/armOrigin AT 22 : ARRAY[1..3] OF REAL := [3(0.0)];
    robot6axis_ctrled1/robot6axis/arm1RowA/overallArmQuatInput AT 6600 : ARRAY[1..4] OF REAL := [4(0.0)];
    robot6axis_ctrled1/robot6axis/arm1RowA/structRotVector AT 113 : ARRAY[1..3] OF REAL := [0.0, 1.0, 0.0];
    robot6axis_ctrled1/robot6axis/arm1RowA/structRotDeg AT 112 : REAL := -90.0;
    robot6axis_ctrled1/robot6axis/arm1RowA/driveRotVector AT 6414 : ARRAY[1..3] OF REAL := [2(0.0), 1.0];
    robot6axis_ctrled1/robot6axis/arm1RowA/driveRotDeg AT 6413 : REAL := 0.0;
    robot6axis_ctrled1/robot6axis/arm1RowA/ownRotDeg AT 6412 : REAL := 0.0;
    robot6axis_ctrled1/robot6axis/arm1RowA/driveResizeLength AT 6411 : REAL := 0.0;
    robot6axis_ctrled1/robot6axis/arm1RowA/functionActive AT 185 : BOOL := false;
    robot6axis_ctrled1/robot6axis/arm1RowA/armExtrem AT 6606 : ARRAY[1..3] OF REAL := [3(0.0)];
    robot6axis_ctrled1/robot6axis/arm1RowA/overallArmRotOutput AT 6611 : ARRAY[1..4] OF REAL := [4(0.0)];
    robot6axis_ctrled1/robot6axis/arm1RowA/productId AT 647 : DINT := -1;
    robot6axis_ctrled1/robot6axis/arm1RowA/status_act_prod AT 709 : DINT := 0;
    robot6axis_ctrled1/robot6axis/arm1RowA/m11 AT 7036 : REAL := 127.321;
    robot6axis_ctrled1/robot6axis/arm1RowA/m12 AT 7037 : REAL := 0.0;
    robot6axis_ctrled1/robot6axis/arm1RowA/m13 AT 7038 : REAL := 0.0;
    robot6axis_ctrled1/robot6axis/arm1RowA/m14 AT 7039 : REAL := 598.055;
    robot6axis_ctrled1/robot6axis/arm1RowA/m21 AT 7040 : REAL := 0.0;
    robot6axis_ctrled1/robot6axis/arm1RowA/m22 AT 7041 : REAL := 1.0;
    robot6axis_ctrled1/robot6axis/arm1RowA/m23 AT 7042 : REAL := 0.0;
    robot6axis_ctrled1/robot6axis/arm1RowA/m24 AT 7043 : REAL := 1.0;
    robot6axis_ctrled1/robot6axis/arm1RowA/m31 AT 7044 : REAL := 0.0;
    robot6axis_ctrled1/robot6axis/arm1RowA/m32 AT 7045 : REAL := 0.0;
    robot6axis_ctrled1/robot6axis/arm1RowA/m33 AT 7046 : REAL := 35.3669;
    robot6axis_ctrled1/robot6axis/arm1RowA/m34 AT 7047 : REAL := 215.827;
    robot6axis_ctrled1/robot6axis/arm1RowA/m41 AT 7048 : REAL := 0.0;
    robot6axis_ctrled1/robot6axis/arm1RowA/m42 AT 7049 : REAL := 0.0;
    robot6axis_ctrled1/robot6axis/arm1RowA/m43 AT 7050 : REAL := 0.0;
    robot6axis_ctrled1/robot6axis/arm1RowA/m44 AT 7051 : REAL := 1.0;
    robot6axis_ctrled1/robot6axis/arm1RowA/armLengthCalc AT 7052 : REAL := 0.0;
    robot6axis_ctrled1/robot6axis/arm1RowA/functionActiveLocale AT 341 : BOOL := false;
    robot6axis_ctrled1/robot6axis/arm1RowA/product_id AT 710 : DINT := -1;
    robot6axis_ctrled1/robot6axis/arm1RowA/arm_id AT 711 : DINT := -1;
    robot6axis_ctrled1/robot6axis/arm1RowA/timeToGripParam AT 7053 : REAL := 0.15;
    robot6axis_ctrled1/robot6axis/arm1RowA/armLength AT 7054 : REAL := 100.0;
    robot6axis_ctrled1/robot6axis/arm1RowA/armWidth AT 7055 : REAL := 200.0;
    robot6axis_ctrled1/robot6axis/arm1RowA/armHeight AT 7056 : REAL := 5.0;
    robot6axis_ctrled1/robot6axis/arm1RowA/armType AT 712 : INT := 0;
    robot6axis_ctrled1/robot6axis/arm1RowB/armOrigin AT 6606 : ARRAY[1..3] OF REAL := [3(0.0)];
    robot6axis_ctrled1/robot6axis/arm1RowB/overallArmQuatInput AT 6611 : ARRAY[1..4] OF REAL := [4(0.0)];
    robot6axis_ctrled1/robot6axis/arm1RowB/structRotVector AT 107 : ARRAY[1..3] OF REAL := [0.0, 1.0, 0.0];
    robot6axis_ctrled1/robot6axis/arm1RowB/structRotDeg AT 106 : REAL := 90.0;
    robot6axis_ctrled1/robot6axis/arm1RowB/driveRotVector AT 6406 : ARRAY[1..3] OF REAL := [2(0.0), 1.0];
    robot6axis_ctrled1/robot6axis/arm1RowB/driveRotDeg AT 6405 : REAL := 0.0;
    robot6axis_ctrled1/robot6axis/arm1RowB/ownRotDeg AT 6404 : REAL := 0.0;
    robot6axis_ctrled1/robot6axis/arm1RowB/driveResizeLength AT 6403 : REAL := 0.0;
    robot6axis_ctrled1/robot6axis/arm1RowB/functionActive AT 21 : BOOL := false;
    robot6axis_ctrled1/robot6axis/arm1RowB/armExtrem AT 6398 : ARRAY[1..3] OF REAL := [3(0.0)];
    robot6axis_ctrled1/robot6axis/arm1RowB/overallArmRotOutput AT 6392 : ARRAY[1..4] OF REAL := [4(0.0)];
    robot6axis_ctrled1/robot6axis/arm1RowB/productId AT 646 : DINT := -1;
    robot6axis_ctrled1/robot6axis/arm1RowB/status_act_prod AT 713 : DINT := 0;
    robot6axis_ctrled1/robot6axis/arm1RowB/m11 AT 7057 : REAL := 127.321;
    robot6axis_ctrled1/robot6axis/arm1RowB/m12 AT 7058 : REAL := 0.0;
    robot6axis_ctrled1/robot6axis/arm1RowB/m13 AT 7059 : REAL := 0.0;
    robot6axis_ctrled1/robot6axis/arm1RowB/m14 AT 7060 : REAL := 594.872;
    robot6axis_ctrled1/robot6axis/arm1RowB/m21 AT 7061 : REAL := 0.0;
    robot6axis_ctrled1/robot6axis/arm1RowB/m22 AT 7062 : REAL := 1.0;
    robot6axis_ctrled1/robot6axis/arm1RowB/m23 AT 7063 : REAL := 0.0;
    robot6axis_ctrled1/robot6axis/arm1RowB/m24 AT 7064 : REAL := 1.0;
    robot6axis_ctrled1/robot6axis/arm1RowB/m31 AT 7065 : REAL := 0.0;
    robot6axis_ctrled1/robot6axis/arm1RowB/m32 AT 7066 : REAL := 0.0;
    robot6axis_ctrled1/robot6axis/arm1RowB/m33 AT 7067 : REAL := 34.6596;
    robot6axis_ctrled1/robot6axis/arm1RowB/m34 AT 7068 : REAL := 163.13;
    robot6axis_ctrled1/robot6axis/arm1RowB/m41 AT 7069 : REAL := 0.0;
    robot6axis_ctrled1/robot6axis/arm1RowB/m42 AT 7070 : REAL := 0.0;
    robot6axis_ctrled1/robot6axis/arm1RowB/m43 AT 7071 : REAL := 0.0;
    robot6axis_ctrled1/robot6axis/arm1RowB/m44 AT 7072 : REAL := 1.0;
    robot6axis_ctrled1/robot6axis/arm1RowB/armLengthCalc AT 7073 : REAL := 0.0;
    robot6axis_ctrled1/robot6axis/arm1RowB/functionActiveLocale AT 342 : BOOL := false;
    robot6axis_ctrled1/robot6axis/arm1RowB/product_id AT 714 : DINT := -1;
    robot6axis_ctrled1/robot6axis/arm1RowB/arm_id AT 715 : DINT := -1;
    robot6axis_ctrled1/robot6axis/arm1RowB/timeToGripParam AT 7074 : REAL := 0.15;
    robot6axis_ctrled1/robot6axis/arm1RowB/armLength AT 7075 : REAL := 50.0;
    robot6axis_ctrled1/robot6axis/arm1RowB/armWidth AT 7076 : REAL := 200.0;
    robot6axis_ctrled1/robot6axis/arm1RowB/armHeight AT 7077 : REAL := 5.0;
    robot6axis_ctrled1/robot6axis/arm1RowB/armType AT 716 : INT := 0;
    conveyors/forwardUp AT 25 : BOOL := false;
    conveyors/backwardUp AT 26 : BOOL := false;
    conveyors/forwardDw AT 27 : BOOL := false;
    conveyors/backwardDw AT 28 : BOOL := false;
    conveyors/ejectBadProd AT 29 : BOOL := false;
    conveyors/presConvUp AT 6 : BOOL := false;
    conveyors/presConvDw AT 7 : BOOL := false;
    conveyors/idRead AT 525 : INT := 0;
    conveyors/mesuredWeight AT 526 : INT := 0;
    conveyors/bpStart AT 8 : BOOL := false;
    conveyors/bpAuto AT 9 : BOOL := false;
    conveyors/bpManu AT 10 : BOOL := false;
    conveyors/bpEmergencyStop AT 11 : BOOL := false;
    conveyors/bpStop AT 12 : BOOL := false;
    conveyors/motConvUp/voltage380 AT 361 : BOOL := true;
    conveyors/motConvUp/cmdSupply AT 360 : BOOL := true;
    conveyors/motConvUp/sensorSupply AT 359 : BOOL := true;
    conveyors/motConvUp/forward AT 25 : BOOL := false;
    conveyors/motConvUp/backward AT 26 : BOOL := false;
    conveyors/motConvUp/forwardFB AT 358 : BOOL := false;
    conveyors/motConvUp/backwardFB AT 357 : BOOL := false;
    conveyors/motConvUp/thermal AT 356 : BOOL := false;
    conveyors/motConvUp/speedVal AT 7120 : REAL := 0.0;
    conveyors/motConvUp/speedPercent AT 7119 : REAL := 0.0;
    conveyors/motConvUp/increment AT 7123 : REAL := 0.0;
    conveyors/motConvUp/memoFwd AT 362 : BOOL := false;
    conveyors/motConvUp/memoBwd AT 363 : BOOL := false;
    conveyors/motConvUp/forwardState AT 364 : BOOL := false;
    conveyors/motConvUp/backwardState AT 365 : BOOL := false;
    conveyors/motConvUp/wantedSpeed AT 7124 : REAL := 0.0;
    conveyors/motConvUp/nominalSpeed AT 7125 : REAL := 50.0;
    conveyors/motConvUp/nominalTime AT 7126 : REAL := 0.5;
    conveyors/motConvUp/thermalLogic AT 366 : BOOL := false;
    conveyors/motConvUp/fwdFbLogic AT 367 : BOOL := true;
    conveyors/motConvUp/bwdFbLogic AT 368 : BOOL := true;
    conveyors/motConvUp/d_locking AT 369 : BOOL := false;
    conveyors/motConvUp/v_d_locking AT 7127 : REAL := 0.0;
    conveyors/motConvUp/d_electrical AT 370 : BOOL := false;
    conveyors/motConvUp/v_d_electrical AT 371 : BOOL := false;
    conveyors/motConvUp/d_backwardFB AT 372 : BOOL := false;
    conveyors/motConvUp/v_d_backwardFB AT 373 : BOOL := false;
    conveyors/motConvUp/d_forwardFB AT 374 : BOOL := false;
    conveyors/motConvUp/v_d_forwardFB AT 375 : BOOL := false;
    conveyors/mtConvDw/voltage380 AT 355 : BOOL := true;
    conveyors/mtConvDw/cmdSupply AT 354 : BOOL := true;
    conveyors/mtConvDw/sensorSupply AT 353 : BOOL := true;
    conveyors/mtConvDw/forward AT 27 : BOOL := false;
    conveyors/mtConvDw/backward AT 28 : BOOL := false;
    conveyors/mtConvDw/forwardFB AT 352 : BOOL := false;
    conveyors/mtConvDw/backwardFB AT 351 : BOOL := false;
    conveyors/mtConvDw/thermal AT 350 : BOOL := false;
    conveyors/mtConvDw/speedVal AT 7121 : REAL := 0.0;
    conveyors/mtConvDw/speedPercent AT 7118 : REAL := 0.0;
    conveyors/mtConvDw/increment AT 7128 : REAL := 0.0;
    conveyors/mtConvDw/memoFwd AT 376 : BOOL := false;
    conveyors/mtConvDw/memoBwd AT 377 : BOOL := false;
    conveyors/mtConvDw/forwardState AT 378 : BOOL := false;
    conveyors/mtConvDw/backwardState AT 379 : BOOL := false;
    conveyors/mtConvDw/wantedSpeed AT 7129 : REAL := 0.0;
    conveyors/mtConvDw/nominalSpeed AT 7130 : REAL := 50.0;
    conveyors/mtConvDw/nominalTime AT 7131 : REAL := 0.05;
    conveyors/mtConvDw/thermalLogic AT 380 : BOOL := false;
    conveyors/mtConvDw/fwdFbLogic AT 381 : BOOL := true;
    conveyors/mtConvDw/bwdFbLogic AT 382 : BOOL := true;
    conveyors/mtConvDw/d_locking AT 383 : BOOL := false;
    conveyors/mtConvDw/v_d_locking AT 7132 : REAL := 0.0;
    conveyors/mtConvDw/d_electrical AT 384 : BOOL := false;
    conveyors/mtConvDw/v_d_electrical AT 385 : BOOL := false;
    conveyors/mtConvDw/d_backwardFB AT 386 : BOOL := false;
    conveyors/mtConvDw/v_d_backwardFB AT 387 : BOOL := false;
    conveyors/mtConvDw/d_forwardFB AT 388 : BOOL := false;
    conveyors/mtConvDw/v_d_forwardFB AT 389 : BOOL := false;
    conveyors/product_creator1/status_act_prod AT 717 : DINT := 0;
    conveyors/product_creator1/m11 AT 7133 : REAL := 30.0619;
    conveyors/product_creator1/m12 AT 7134 : REAL := 0.0;
    conveyors/product_creator1/m13 AT 7135 : REAL := 0.0;
    conveyors/product_creator1/m14 AT 7136 : REAL := 1246.07;
    conveyors/product_creator1/m21 AT 7137 : REAL := 0.0;
    conveyors/product_creator1/m22 AT 7138 : REAL := 200.0;
    conveyors/product_creator1/m23 AT 7139 : REAL := 0.0;
    conveyors/product_creator1/m24 AT 7140 : REAL := 615.0;
    conveyors/product_creator1/m31 AT 7141 : REAL := 0.0;
    conveyors/product_creator1/m32 AT 7142 : REAL := 0.0;
    conveyors/product_creator1/m33 AT 7143 : REAL := 99.9116;
    conveyors/product_creator1/m34 AT 7144 : REAL := 428.912;
    conveyors/product_creator1/m41 AT 7145 : REAL := 0.0;
    conveyors/product_creator1/m42 AT 7146 : REAL := 0.0;
    conveyors/product_creator1/m43 AT 7147 : REAL := 0.0;
    conveyors/product_creator1/m44 AT 7148 : REAL := 1.0;
    conveyors/product_creator1/pbCreation AT 390 : BOOL := false;
    conveyors/product_creator1/productPresence AT 391 : BOOL := false;
    conveyors/product_creator1/idProd AT 718 : DINT := 0;
    conveyors/product_creator1/cntProd AT 719 : DINT := 0;
    conveyors/product_creator1/waitingTime AT 7149 : REAL := 10.0;
    conveyors/product_creator1/oldIdProd AT 720 : DINT := 0;
    conveyors/product_creator1/empty1 AT 392 : BOOL := false;
    conveyors/product_creator1/empty2 AT 393 : BOOL := false;
    conveyors/product_creator1/empty3 AT 394 : BOOL := false;
    conveyors/product_creator1/empty4 AT 395 : BOOL := false;
    conveyors/product_creator1/empty5 AT 396 : BOOL := false;
    conveyors/product_creator1/empty6 AT 397 : BOOL := false;
    conveyors/product_creator1/empty7 AT 398 : BOOL := false;
    conveyors/product_creator1/empty8 AT 399 : BOOL := false;
    conveyors/product_creator1/gravitySpeed AT 7150 : REAL := 0.1;
    conveyors/product_creator1/nbProdToCreate AT 721 : INT := 1;
    conveyors/product_creator1/pulsedMode AT 400 : BOOL := false;
    conveyors/product_creator1/pulseTime AT 7151 : REAL := 8.0;
    conveyors/product_creator1/alignProductsToZ AT 401 : BOOL := true;
    conveyors/product_creator1/alignProductsToY AT 402 : BOOL := false;
    conveyors/product_creator1/alignProductsToX AT 403 : BOOL := false;
    conveyors/product_killer1/status_act_prod AT 722 : DINT := 0;
    conveyors/product_killer1/m11 AT 7152 : REAL := 26.5252;
    conveyors/product_killer1/m12 AT 7153 : REAL := 0.0;
    conveyors/product_killer1/m13 AT 7154 : REAL := 0.0;
    conveyors/product_killer1/m14 AT 7155 : REAL := 698.983;
    conveyors/product_killer1/m21 AT 7156 : REAL := 0.0;
    conveyors/product_killer1/m22 AT 7157 : REAL := 35.809;
    conveyors/product_killer1/m23 AT 7158 : REAL := 0.0;
    conveyors/product_killer1/m24 AT 7159 : REAL := 1244.74;
    conveyors/product_killer1/m31 AT 7160 : REAL := 0.0;
    conveyors/product_killer1/m32 AT 7161 : REAL := 0.0;
    conveyors/product_killer1/m33 AT 7162 : REAL := 38.9036;
    conveyors/product_killer1/m34 AT 7163 : REAL := 662.776;
    conveyors/product_killer1/m41 AT 7164 : REAL := 0.0;
    conveyors/product_killer1/m42 AT 7165 : REAL := 0.0;
    conveyors/product_killer1/m43 AT 7166 : REAL := 0.0;
    conveyors/product_killer1/m44 AT 7167 : REAL := 1.0;
    conveyors/product_killer1/isActive AT 404 : BOOL := true;
